C07267=1135.788,-43.089,-47.280,179.177,6.196,149.362
C07268=1135.793,-43.339,-47.268,179.175,6.195,149.362
C07269=1135.798,-43.589,-47.258,179.172,6.194,149.363
C07270=1135.804,-43.838,-47.246,179.170,6.194,149.363
C07271=1135.809,-44.088,-47.235,179.168,6.193,149.364
C07272=1135.814,-44.337,-47.224,179.165,6.193,149.364
C07273=1135.820,-44.587,-47.213,179.163,6.192,149.365
C07274=1135.825,-44.837,-47.202,179.160,6.191,149.366
C07275=1135.829,-45.086,-47.190,179.158,6.191,149.366
C07276=1135.836,-45.336,-47.180,179.156,6.190,149.367
C07277=1135.840,-45.586,-47.168,179.153,6.189,149.367
C07278=1135.845,-45.835,-47.157,179.151,6.189,149.368
C07279=1135.851,-46.085,-47.146,179.149,6.188,149.368
C07280=1135.856,-46.335,-47.135,179.147,6.187,149.369
C07281=1135.861,-46.585,-47.124,179.144,6.187,149.369
C07282=1135.867,-46.834,-47.113,179.143,6.187,149.370
C07283=1135.872,-47.084,-47.102,179.140,6.186,149.370
C07284=1135.877,-47.334,-47.091,179.138,6.186,149.371
C07285=1135.883,-47.584,-47.079,179.136,6.185,149.371
C07286=1135.887,-47.833,-47.068,179.133,6.184,149.372
C07287=1135.893,-48.083,-47.058,179.131,6.183,149.372
C07288=1135.898,-48.333,-47.046,179.129,6.183,149.373
C07289=1135.903,-48.583,-47.036,179.126,6.182,149.374
C07290=1135.909,-48.832,-47.025,179.124,6.181,149.374
C07291=1135.913,-49.081,-47.013,179.121,6.181,149.375
C07292=1135.919,-49.332,-47.002,179.119,6.180,149.375
C07293=1135.924,-49.581,-46.991,179.117,6.179,149.376
C07294=1135.929,-49.831,-46.981,179.115,6.179,149.376
C07295=1135.935,-50.080,-46.970,179.113,6.179,149.377
C07296=1135.940,-50.331,-46.959,179.111,6.178,149.377
C07297=1135.946,-50.602,-46.946,179.108,6.177,149.378
C07298=1135.952,-50.872,-46.935,179.105,6.176,149.379
C07299=1135.957,-51.143,-46.923,179.103,6.176,149.379
C07300=1135.963,-51.413,-46.911,179.100,6.175,149.380
C07301=1135.968,-51.663,-46.900,179.098,6.174,149.380
C07302=1135.973,-51.913,-46.889,179.097,6.174,149.381
C07303=1135.979,-52.162,-46.879,179.094,6.174,149.381
C07304=1135.984,-52.412,-46.867,179.092,6.173,149.382
C07305=1135.990,-52.662,-46.857,179.090,6.172,149.382
C07306=1135.995,-52.912,-46.846,179.087,6.172,149.383
C07307=1136.000,-53.161,-46.835,179.085,6.171,149.384
C07308=1136.005,-53.411,-46.825,179.082,6.171,149.384
C07309=1136.011,-53.660,-46.813,179.080,6.170,149.385
C07310=1136.016,-53.911,-46.803,179.078,6.169,149.385
C07311=1136.021,-54.160,-46.792,179.075,6.169,149.386
C07312=1136.026,-54.410,-46.781,179.074,6.169,149.386
C07313=1136.031,-54.660,-46.770,179.072,6.168,149.387
C07314=1136.037,-54.909,-46.760,179.069,6.167,149.387
C07315=1136.042,-55.159,-46.749,179.067,6.167,149.388
C07316=1136.048,-55.408,-46.737,179.065,6.166,149.388
C07317=1136.053,-55.659,-46.727,179.062,6.165,149.389
C07318=1136.058,-55.908,-46.717,179.060,6.165,149.390
C07319=1136.063,-56.158,-46.705,179.058,6.164,149.390
C07320=1136.069,-56.407,-46.695,179.056,6.164,149.390
C07321=1136.074,-56.658,-46.685,179.054,6.163,149.391
C07322=1136.079,-56.907,-46.674,179.051,6.163,149.392
C07323=1136.084,-57.157,-46.663,179.049,6.162,149.392
C07324=1136.089,-57.406,-46.653,179.047,6.161,149.393
C07325=1136.094,-57.656,-46.642,179.045,6.161,149.393
C07326=1136.100,-57.906,-46.631,179.042,6.160,149.394
C07327=1136.105,-58.156,-46.620,179.040,6.159,149.394
C07328=1136.111,-58.405,-46.609,179.038,6.159,149.395
C07329=1136.116,-58.655,-46.599,179.035,6.159,149.395
C07330=1136.121,-58.905,-46.589,179.033,6.158,149.396
C07331=1136.126,-59.155,-46.578,179.031,6.157,149.396
C07332=1136.132,-59.404,-46.567,179.029,6.157,149.397
C07333=1136.137,-59.654,-46.557,179.026,6.156,149.398
C07334=1136.142,-59.904,-46.546,179.024,6.156,149.398
C07335=1136.148,-60.153,-46.536,179.022,6.156,149.399
C07336=1136.153,-60.403,-46.525,179.020,6.155,149.399
C07337=1136.158,-60.652,-46.515,179.018,6.154,149.400
C07338=1136.163,-60.903,-46.504,179.015,6.154,149.400
C07339=1136.169,-61.152,-46.494,179.013,6.153,149.401
C07340=1136.174,-61.403,-46.483,179.011,6.152,149.401
C07341=1136.179,-61.651,-46.472,179.008,6.152,149.402
C07342=1136.185,-61.901,-46.462,179.007,6.152,149.402
C07343=1136.190,-62.151,-46.451,179.004,6.151,149.403
C07344=1136.195,-62.401,-46.441,179.002,6.150,149.403
C07345=1136.200,-62.651,-46.431,179.000,6.150,149.404
C07346=1136.205,-62.900,-46.420,178.997,6.149,149.405
C07347=1136.211,-63.149,-46.410,178.995,6.148,149.405
C07348=1136.216,-63.400,-46.399,178.994,6.148,149.406
C07349=1136.222,-63.649,-46.389,178.991,6.148,149.406
C07350=1136.227,-63.900,-46.378,178.989,6.147,149.407
C07351=1136.232,-64.149,-46.368,178.987,6.146,149.407
C07352=1136.238,-64.399,-46.358,178.984,6.146,149.408
C07353=1136.243,-64.649,-46.347,178.982,6.145,149.408
C07354=1136.248,-64.898,-46.338,178.980,6.145,149.409
C07355=1136.252,-65.148,-46.326,178.978,6.145,149.409
C07356=1136.258,-65.397,-46.316,178.976,6.144,149.410
C07357=1136.264,-65.647,-46.306,178.974,6.143,149.410
C07358=1136.269,-65.897,-46.295,178.971,6.143,149.411
C07359=1136.274,-66.147,-46.285,178.969,6.142,149.411
C07360=1136.280,-66.396,-46.275,178.967,6.142,149.412
C07361=1136.285,-66.646,-46.264,178.965,6.141,149.412
C07362=1136.290,-66.896,-46.254,178.962,6.141,149.413
C07363=1136.296,-67.145,-46.244,178.960,6.140,149.414
C07364=1136.301,-67.396,-46.233,178.958,6.139,149.414
C07365=1136.306,-67.645,-46.224,178.956,6.139,149.415
C07366=1136.311,-67.894,-46.213,178.954,6.139,149.415
C07367=1136.316,-68.145,-46.203,178.951,6.138,149.416
C07368=1136.322,-68.394,-46.193,178.949,6.137,149.416
C07369=1136.328,-68.644,-46.182,178.947,6.137,149.417
C07370=1136.333,-68.894,-46.172,178.945,6.136,149.417
C07371=1136.338,-69.144,-46.162,178.943,6.136,149.418
C07372=1136.343,-69.393,-46.152,178.941,6.136,149.418
C07373=1136.348,-69.643,-46.142,178.938,6.135,149.419
C07374=1136.354,-69.893,-46.131,178.936,6.134,149.419
C07375=1136.359,-70.142,-46.121,178.933,6.134,149.420
C07376=1136.364,-70.392,-46.111,178.932,6.134,149.421
C07377=1136.370,-70.642,-46.100,178.930,6.133,149.421
C07378=1136.375,-70.891,-46.091,178.928,6.132,149.422
C07379=1136.380,-71.141,-46.081,178.925,6.131,149.422
C07380=1136.386,-71.392,-46.071,178.923,6.132,149.423
C07381=1136.391,-71.641,-46.060,178.921,6.131,149.423
C07382=1136.397,-71.891,-46.050,178.919,6.130,149.424
C07383=1136.401,-72.141,-46.040,178.917,6.129,149.424
C07384=1136.407,-72.390,-46.030,178.914,6.129,149.425
C07385=1136.412,-72.640,-46.020,178.912,6.129,149.425
C07386=1136.418,-72.889,-46.010,178.910,6.128,149.426
C07387=1136.422,-73.139,-46.000,178.908,6.128,149.426
C07388=1136.428,-73.389,-45.990,178.906,6.127,149.427
C07389=1136.434,-73.639,-45.980,178.903,6.126,149.428
C07390=1136.439,-73.888,-45.970,178.902,6.127,149.428
C07391=1136.444,-74.139,-45.959,178.899,6.126,149.428
C07392=1136.449,-74.388,-45.950,178.897,6.125,149.429
C07393=1136.455,-74.637,-45.939,178.895,6.124,149.429
C07394=1136.461,-74.888,-45.930,178.893,6.125,149.430
C07395=1136.465,-75.138,-45.920,178.891,6.124,149.431
C07396=1136.470,-75.387,-45.910,178.889,6.123,149.431
C07397=1136.476,-75.637,-45.899,178.886,6.122,149.432
C07398=1136.482,-75.886,-45.889,178.884,6.122,149.432
C07399=1136.487,-76.136,-45.880,178.882,6.122,149.433
C07400=1136.492,-76.386,-45.870,178.880,6.121,149.433
C07401=1136.498,-76.657,-45.859,178.878,6.120,149.434
C07402=1136.504,-76.929,-45.848,178.875,6.120,149.434
C07403=1136.509,-77.200,-45.837,178.873,6.119,149.435
C07404=1136.516,-77.472,-45.827,178.871,6.119,149.435
C07405=1136.520,-77.722,-45.817,178.869,6.119,149.436
C07406=1136.526,-77.971,-45.807,178.866,6.118,149.437
C07407=1136.531,-78.221,-45.797,178.864,6.118,149.437
C07408=1136.537,-78.471,-45.788,178.862,6.117,149.438
C07409=1136.542,-78.720,-45.777,178.860,6.117,149.438
C07410=1136.548,-78.970,-45.767,178.858,6.116,149.439
C07411=1136.552,-79.220,-45.758,178.856,6.116,149.439
C07412=1136.558,-79.470,-45.748,178.853,6.115,149.440
C07413=1136.563,-79.719,-45.738,178.852,6.115,149.440
C07414=1136.569,-79.969,-45.729,178.850,6.114,149.441
C07415=1136.574,-80.219,-45.718,178.847,6.113,149.441
C07416=1136.580,-80.468,-45.708,178.845,6.113,149.442
C07417=1136.584,-80.719,-45.699,178.843,6.113,149.442
C07418=1136.590,-80.969,-45.689,178.841,6.112,149.443
C07419=1136.595,-81.218,-45.679,178.839,6.112,149.443
C07420=1136.601,-81.468,-45.670,178.836,6.111,149.444
C07421=1136.606,-81.717,-45.659,178.835,6.111,149.444
C07422=1136.612,-81.967,-45.651,178.832,6.110,149.445
C07423=1136.617,-82.218,-45.640,178.830,6.110,149.446
C07424=1136.621,-82.467,-45.630,178.828,6.109,149.446
C07425=1136.627,-82.717,-45.621,178.826,6.109,149.447
C07426=1136.632,-82.966,-45.611,178.824,6.108,149.447
C07427=1136.638,-83.216,-45.602,178.822,6.107,149.447
C07428=1136.644,-83.466,-45.592,178.820,6.108,149.448
C07429=1136.649,-83.716,-45.583,178.818,6.107,149.449
C07430=1136.654,-83.965,-45.572,178.815,6.106,149.449
C07431=1136.659,-84.215,-45.563,178.813,6.106,149.450
C07432=1136.665,-84.465,-45.553,178.812,6.106,149.450
C07433=1136.669,-84.715,-45.543,178.809,6.105,149.451
C07434=1136.675,-84.965,-45.534,178.807,6.105,149.451
C07435=1136.680,-85.214,-45.524,178.805,6.104,149.452
C07436=1136.686,-85.464,-45.515,178.803,6.104,149.452
C07437=1136.691,-85.713,-45.505,178.801,6.103,149.453
C07438=1136.697,-85.964,-45.496,178.799,6.102,149.453
C07439=1136.702,-86.213,-45.486,178.797,6.102,149.454
C07440=1136.708,-86.463,-45.477,178.794,6.102,149.454
C07441=1136.713,-86.712,-45.467,178.792,6.101,149.455
C07442=1136.718,-86.963,-45.457,178.790,6.100,149.455
C07443=1136.723,-87.212,-45.447,178.788,6.100,149.456
C07444=1136.729,-87.462,-45.438,178.786,6.100,149.456
C07445=1136.733,-87.712,-45.428,178.784,6.099,149.457
C07446=1136.739,-87.962,-45.419,178.782,6.099,149.458
C07447=1136.745,-88.212,-45.410,178.780,6.099,149.458
C07448=1136.749,-88.461,-45.400,178.777,6.098,149.459
C07449=1136.755,-88.711,-45.391,178.776,6.098,149.459
C07450=1136.760,-88.960,-45.381,178.774,6.097,149.460
C07451=1136.766,-89.210,-45.372,178.771,6.096,149.460
C07452=1136.771,-89.460,-45.362,178.769,6.096,149.460
C07453=1136.777,-89.710,-45.353,178.767,6.096,149.461
C07454=1136.782,-89.960,-45.344,178.765,6.095,149.462
C07455=1136.788,-90.209,-45.334,178.763,6.095,149.462
C07456=1136.793,-90.459,-45.325,178.761,6.095,149.463
C07457=1136.798,-90.708,-45.315,178.759,6.094,149.463
C07458=1136.803,-90.959,-45.306,178.757,6.093,149.464
C07459=1136.809,-91.208,-45.297,178.755,6.093,149.464
C07460=1136.814,-91.458,-45.286,178.753,6.093,149.465
C07461=1136.819,-91.708,-45.278,178.750,6.092,149.465
C07462=1136.825,-91.958,-45.269,178.749,6.092,149.466
C07463=1136.830,-92.207,-45.258,178.747,6.091,149.466
C07464=1136.835,-92.457,-45.250,178.744,6.091,149.467
C07465=1136.841,-92.707,-45.241,178.743,6.091,149.467
C07466=1136.846,-92.956,-45.230,178.741,6.090,149.468
C07467=1136.851,-93.206,-45.222,178.738,6.089,149.468
C07468=1136.857,-93.456,-45.212,178.736,6.090,149.469
C07469=1136.862,-93.706,-45.203,178.734,6.089,149.469
C07470=1136.867,-93.955,-45.194,178.732,6.088,149.470
C07471=1136.873,-94.206,-45.184,178.730,6.088,149.470
C07472=1136.878,-94.456,-45.175,178.728,6.087,149.471
C07473=1136.883,-94.705,-45.166,178.726,6.087,149.471
C07474=1136.889,-94.955,-45.156,178.724,6.087,149.472
C07475=1136.894,-95.205,-45.147,178.722,6.086,149.473
C07476=1136.899,-95.455,-45.138,178.719,6.085,149.473
C07477=1136.905,-95.704,-45.128,178.718,6.085,149.474
C07478=1136.910,-95.954,-45.119,178.716,6.085,149.474
C07479=1136.915,-96.204,-45.110,178.713,6.084,149.474
C07480=1136.920,-96.454,-45.101,178.712,6.084,149.475
C07481=1136.926,-96.704,-45.092,178.710,6.083,149.475
C07482=1136.931,-96.953,-45.082,178.707,6.083,149.476
C07483=1136.936,-97.203,-45.073,178.706,6.083,149.476
C07484=1136.942,-97.453,-45.064,178.703,6.082,149.477
C07485=1136.948,-97.702,-45.055,178.701,6.081,149.478
C07486=1136.953,-97.952,-45.046,178.699,6.081,149.478
C07487=1136.958,-98.201,-45.037,178.697,6.081,149.479
C07488=1136.964,-98.452,-45.027,178.695,6.080,149.479
C07489=1136.969,-98.701,-45.018,178.693,6.080,149.480
C07490=1136.974,-98.951,-45.010,178.691,6.079,149.480
C07491=1136.980,-99.201,-45.000,178.689,6.079,149.481
C07492=1136.985,-99.451,-44.991,178.687,6.079,149.481
C07493=1136.991,-99.701,-44.982,178.685,6.078,149.482
C07494=1136.996,-99.951,-44.973,178.683,6.077,149.482
C07495=1137.001,-100.200,-44.963,178.681,6.077,149.483
C07496=1137.007,-100.450,-44.955,178.679,6.077,149.483
C07497=1137.012,-100.699,-44.946,178.677,6.077,149.484
C07498=1137.017,-100.949,-44.937,178.675,6.076,149.484
C07499=1137.023,-101.199,-44.928,178.673,6.075,149.485
C07500=1137.029,-101.449,-44.918,178.671,6.075,149.485
C07501=1137.034,-101.699,-44.910,178.669,6.075,149.486
C07502=1137.039,-101.949,-44.901,178.667,6.074,149.486
C07503=1137.044,-102.199,-44.892,178.665,6.074,149.487
C07504=1137.049,-102.449,-44.883,178.663,6.074,149.487
C07505=1137.055,-102.720,-44.873,178.660,6.073,149.488
C07506=1137.062,-102.993,-44.863,178.659,6.073,149.488
C07507=1137.067,-103.265,-44.853,178.657,6.072,149.489
C07508=1137.073,-103.537,-44.843,178.654,6.072,149.489
C07509=1137.078,-103.787,-44.834,178.652,6.071,149.490
C07510=1137.083,-104.037,-44.825,178.650,6.071,149.490
C07511=1137.089,-104.286,-44.817,178.648,6.070,149.491
C07512=1137.094,-104.536,-44.808,178.646,6.070,149.491
C07513=1137.100,-104.786,-44.799,178.644,6.070,149.492
C07514=1137.105,-105.036,-44.789,178.642,6.069,149.492
C07515=1137.111,-105.286,-44.781,178.640,6.069,149.493
C07516=1137.116,-105.536,-44.772,178.638,6.068,149.493
C07517=1137.121,-105.786,-44.763,178.636,6.067,149.494
C07518=1137.127,-106.035,-44.754,178.634,6.067,149.494
C07519=1137.132,-106.285,-44.745,178.632,6.067,149.495
C07520=1137.137,-106.534,-44.736,178.631,6.067,149.495
C07521=1137.142,-106.784,-44.728,178.628,6.066,149.496
C07522=1137.147,-107.034,-44.719,178.626,6.066,149.497
C07523=1137.153,-107.283,-44.710,178.624,6.066,149.497
C07524=1137.159,-107.533,-44.701,178.622,6.065,149.497
C07525=1137.165,-107.784,-44.692,178.620,6.065,149.498
C07526=1137.170,-108.034,-44.684,178.618,6.064,149.498
C07527=1137.175,-108.284,-44.675,178.616,6.063,149.499
C07528=1137.181,-108.533,-44.666,178.614,6.063,149.499
C07529=1137.186,-108.783,-44.657,178.612,6.063,149.500
C07530=1137.191,-109.032,-44.648,178.610,6.063,149.500
C07531=1137.196,-109.282,-44.639,178.608,6.062,149.501
C07532=1137.201,-109.532,-44.631,178.606,6.061,149.501
C07533=1137.207,-109.781,-44.622,178.604,6.061,149.502
C07534=1137.213,-110.032,-44.614,178.602,6.061,149.502
C07535=1137.218,-110.282,-44.605,178.601,6.061,149.503
C07536=1137.223,-110.531,-44.596,178.598,6.060,149.503
C07537=1137.229,-110.781,-44.588,178.597,6.060,149.504
C07538=1137.234,-111.030,-44.579,178.595,6.059,149.504
C07539=1137.239,-111.280,-44.570,178.592,6.058,149.505
C07540=1137.244,-111.530,-44.561,178.590,6.059,149.506
C07541=1137.250,-111.780,-44.553,178.588,6.058,149.506
C07542=1137.255,-112.030,-44.544,178.587,6.058,149.506
C07543=1137.261,-112.280,-44.535,178.584,6.057,149.507
C07544=1137.266,-112.530,-44.526,178.582,6.057,149.507
C07545=1137.271,-112.779,-44.518,178.581,6.057,149.508
C07546=1137.277,-113.029,-44.510,178.578,6.056,149.508
C07547=1137.282,-113.279,-44.501,178.577,6.056,149.509
C07548=1137.287,-113.529,-44.492,178.575,6.055,149.509
C07549=1137.293,-113.778,-44.483,178.573,6.055,149.510
C07550=1137.299,-114.028,-44.475,178.571,6.055,149.510
C07551=1137.304,-114.278,-44.466,178.569,6.054,149.511
C07552=1137.309,-114.527,-44.458,178.567,6.054,149.511
C07553=1137.315,-114.777,-44.449,178.565,6.053,149.512
C07554=1137.320,-115.028,-44.441,178.563,6.053,149.512
C07555=1137.325,-115.278,-44.432,178.561,6.052,149.513
C07556=1137.331,-115.527,-44.423,178.559,6.052,149.513
C07557=1137.336,-115.777,-44.414,178.557,6.052,149.514
C07558=1137.342,-116.027,-44.406,178.555,6.051,149.514
C07559=1137.347,-116.276,-44.398,178.553,6.051,149.515
C07560=1137.353,-116.526,-44.389,178.551,6.050,149.515
C07561=1137.358,-116.777,-44.380,178.550,6.050,149.516
C07562=1137.364,-117.026,-44.372,178.547,6.050,149.516
C07563=1137.369,-117.276,-44.363,178.546,6.050,149.517
C07564=1137.374,-117.526,-44.355,178.544,6.049,149.517
C07565=1137.380,-117.775,-44.347,178.542,6.049,149.518
C07566=1137.385,-118.025,-44.338,178.540,6.048,149.518
C07567=1137.390,-118.275,-44.330,178.538,6.047,149.519
C07568=1137.396,-118.524,-44.321,178.536,6.047,149.519
C07569=1137.401,-118.774,-44.312,178.534,6.047,149.520
C07570=1137.407,-119.025,-44.304,178.532,6.047,149.520
C07571=1137.412,-119.274,-44.296,178.530,6.046,149.521
C07572=1137.417,-119.524,-44.287,178.529,6.046,149.521
C07573=1137.422,-119.774,-44.279,178.526,6.045,149.522
C07574=1137.428,-120.023,-44.271,178.525,6.045,149.522
C07575=1137.433,-120.273,-44.262,178.523,6.045,149.523
C07576=1137.439,-120.523,-44.254,178.521,6.045,149.523
C07577=1137.444,-120.772,-44.245,178.519,6.044,149.524
C07578=1137.450,-121.023,-44.237,178.517,6.043,149.524
C07579=1137.456,-121.272,-44.228,178.515,6.043,149.525
C07580=1137.460,-121.522,-44.221,178.513,6.042,149.525
C07581=1137.466,-121.772,-44.212,178.511,6.042,149.525
C07582=1137.471,-122.021,-44.203,178.509,6.042,149.526
C07583=1137.477,-122.272,-44.195,178.507,6.042,149.526
C07584=1137.482,-122.522,-44.186,178.505,6.041,149.527
C07585=1137.487,-122.771,-44.179,178.504,6.041,149.527
C07586=1137.492,-123.021,-44.170,178.501,6.040,149.528
C07587=1137.499,-123.271,-44.162,178.500,6.040,149.528
C07588=1137.504,-123.520,-44.153,178.498,6.040,149.529
C07589=1137.509,-123.771,-44.145,178.496,6.040,149.529
C07590=1137.514,-124.020,-44.137,178.494,6.039,149.530
C07591=1137.520,-124.270,-44.129,178.492,6.039,149.530
C07592=1137.525,-124.519,-44.121,178.490,6.038,149.531
C07593=1137.531,-124.770,-44.112,178.488,6.038,149.531
C07594=1137.536,-125.020,-44.103,178.486,6.038,149.532
C07595=1137.541,-125.269,-44.096,178.484,6.037,149.532
C07596=1137.547,-125.519,-44.087,178.482,6.037,149.533
C07597=1137.553,-125.769,-44.080,178.481,6.036,149.533
C07598=1137.558,-126.019,-44.071,178.479,6.036,149.534
C07599=1137.563,-126.269,-44.063,178.477,6.035,149.534
C07600=1137.568,-126.518,-44.055,178.475,6.035,149.535
C07601=1137.574,-126.768,-44.046,178.473,6.034,149.535
C07602=1137.580,-127.018,-44.038,178.471,6.034,149.535
C07603=1137.584,-127.268,-44.030,178.469,6.034,149.536
C07604=1137.590,-127.518,-44.022,178.468,6.034,149.536
C07605=1137.596,-127.767,-44.014,178.465,6.033,149.537
C07606=1137.601,-128.017,-44.006,178.464,6.033,149.537
C07607=1137.606,-128.267,-43.997,178.462,6.032,149.538
C07608=1137.612,-128.516,-43.990,178.460,6.032,149.538
C07609=1137.190,-128.528,-44.033,178.456,6.036,149.540
C07610=1137.186,-128.278,-44.041,178.458,6.036,149.540
C07611=1137.180,-128.029,-44.049,178.460,6.036,149.539
C07612=1137.174,-127.778,-44.058,178.462,6.037,149.539
C07613=1137.169,-127.528,-44.066,178.464,6.037,149.538
C07614=1137.164,-127.279,-44.074,178.466,6.038,149.538
C07615=1137.158,-127.029,-44.082,178.468,6.038,149.537
C07616=1137.153,-126.780,-44.090,178.470,6.038,149.537
C07617=1137.147,-126.529,-44.099,178.471,6.038,149.536
C07618=1137.142,-126.280,-44.107,178.474,6.039,149.536
C07619=1137.137,-126.030,-44.115,178.475,6.039,149.535
C07620=1137.132,-125.780,-44.124,178.477,6.040,149.535
C07621=1137.125,-125.530,-44.131,178.479,6.040,149.534
C07622=1137.121,-125.281,-44.140,178.481,6.041,149.534
C07623=1137.115,-125.031,-44.148,178.483,6.040,149.533
C07624=1137.110,-124.780,-44.156,178.485,6.041,149.533
C07625=1137.104,-124.531,-44.164,178.487,6.042,149.532
C07626=1137.099,-124.281,-44.172,178.489,6.042,149.532
C07627=1137.094,-124.031,-44.181,178.491,6.043,149.531
C07628=1137.088,-123.782,-44.189,178.493,6.043,149.531
C07629=1137.083,-123.532,-44.198,178.494,6.044,149.531
C07630=1137.077,-123.282,-44.206,178.496,6.044,149.530
C07631=1137.072,-123.032,-44.214,178.498,6.044,149.530
C07632=1137.067,-122.782,-44.223,178.500,6.044,149.529
C07633=1137.061,-122.533,-44.230,178.502,6.045,149.529
C07634=1137.056,-122.283,-44.239,178.504,6.045,149.528
C07635=1137.050,-122.033,-44.247,178.506,6.046,149.528
C07636=1137.045,-121.784,-44.255,178.507,6.046,149.527
C07637=1137.040,-121.533,-44.264,178.510,6.047,149.527
C07638=1137.034,-121.284,-44.272,178.511,6.046,149.526
C07639=1137.029,-121.034,-44.281,178.513,6.047,149.526
C07640=1137.023,-120.784,-44.289,178.516,6.048,149.525
C07641=1137.018,-120.534,-44.298,178.517,6.048,149.525
C07642=1137.013,-120.284,-44.305,178.519,6.049,149.524
C07643=1137.008,-120.034,-44.314,178.521,6.049,149.524
C07644=1137.002,-119.785,-44.323,178.523,6.049,149.523
C07645=1136.996,-119.535,-44.331,178.525,6.049,149.523
C07646=1136.991,-119.286,-44.339,178.527,6.050,149.522
C07647=1136.985,-119.035,-44.348,178.528,6.050,149.522
C07648=1136.980,-118.785,-44.357,178.531,6.051,149.521
C07649=1136.975,-118.536,-44.364,178.532,6.051,149.521
C07650=1136.969,-118.286,-44.373,178.534,6.051,149.520
C07651=1136.964,-118.036,-44.382,178.537,6.052,149.520
C07652=1136.959,-117.787,-44.390,178.538,6.052,149.519
C07653=1136.953,-117.537,-44.398,178.540,6.053,149.519
C07654=1136.948,-117.287,-44.407,178.542,6.053,149.519
C07655=1136.942,-117.038,-44.416,178.544,6.054,149.518
C07656=1136.937,-116.787,-44.424,178.546,6.054,149.518
C07657=1136.932,-116.537,-44.433,178.548,6.054,149.517
C07658=1136.926,-116.287,-44.442,178.550,6.054,149.517
C07659=1136.920,-116.038,-44.449,178.552,6.055,149.516
C07660=1136.916,-115.788,-44.458,178.554,6.056,149.516
C07661=1136.911,-115.538,-44.467,178.556,6.056,149.515
C07662=1136.905,-115.289,-44.475,178.558,6.056,149.515
C07663=1136.899,-115.039,-44.483,178.559,6.056,149.514
C07664=1136.894,-114.789,-44.492,178.562,6.057,149.514
C07665=1136.889,-114.540,-44.501,178.563,6.057,149.513
C07666=1136.883,-114.289,-44.509,178.565,6.058,149.513
C07667=1136.878,-114.039,-44.518,178.568,6.059,149.512
C07668=1136.873,-113.789,-44.527,178.569,6.059,149.512
C07669=1136.867,-113.540,-44.535,178.571,6.059,149.511
C07670=1136.861,-113.290,-44.544,178.573,6.059,149.511
C07671=1136.856,-113.040,-44.552,178.575,6.060,149.510
C07672=1136.851,-112.791,-44.561,178.577,6.060,149.510
C07673=1136.845,-112.541,-44.570,178.579,6.061,149.509
C07674=1136.840,-112.291,-44.579,178.581,6.061,149.509
C07675=1136.835,-112.041,-44.587,178.583,6.061,149.508
C07676=1136.829,-111.791,-44.595,178.585,6.062,149.508
C07677=1136.824,-111.542,-44.604,178.587,6.062,149.507
C07678=1136.819,-111.292,-44.613,178.589,6.062,149.507
C07679=1136.813,-111.042,-44.622,178.591,6.062,149.506
C07680=1136.808,-110.793,-44.631,178.593,6.063,149.506
C07681=1136.802,-110.542,-44.639,178.595,6.064,149.505
C07682=1136.797,-110.292,-44.648,178.597,6.064,149.505
C07683=1136.792,-110.043,-44.657,178.599,6.065,149.504
C07684=1136.786,-109.793,-44.665,178.601,6.065,149.504
C07685=1136.781,-109.544,-44.674,178.603,6.065,149.503
C07686=1136.776,-109.294,-44.683,178.605,6.066,149.503
C07687=1136.771,-109.044,-44.692,178.607,6.066,149.502
C07688=1136.765,-108.793,-44.700,178.609,6.067,149.502
C07689=1136.759,-108.544,-44.709,178.610,6.067,149.501
C07690=1136.753,-108.294,-44.718,178.613,6.067,149.501
C07691=1136.748,-108.044,-44.727,178.615,6.068,149.500
C07692=1136.743,-107.794,-44.736,178.616,6.068,149.500
C07693=1136.737,-107.545,-44.744,178.619,6.069,149.499
C07694=1136.732,-107.295,-44.753,178.620,6.069,149.499
C07695=1136.727,-107.046,-44.762,178.622,6.070,149.498
C07696=1136.722,-106.796,-44.771,178.625,6.070,149.498
C07697=1136.717,-106.546,-44.780,178.626,6.070,149.497
C07698=1136.712,-106.296,-44.789,178.629,6.071,149.497
C07699=1136.706,-106.047,-44.797,178.630,6.071,149.496
C07700=1136.700,-105.797,-44.807,178.633,6.071,149.496
C07701=1136.695,-105.547,-44.816,178.635,6.072,149.495
C07702=1136.690,-105.297,-44.825,178.636,6.072,149.495
C07703=1136.684,-105.047,-44.834,178.639,6.073,149.494
C07704=1136.679,-104.797,-44.842,178.641,6.074,149.494
C07705=1136.673,-104.548,-44.850,178.642,6.074,149.493
C07706=1136.668,-104.298,-44.859,178.645,6.074,149.493
C07707=1136.663,-104.048,-44.869,178.646,6.074,149.492
C07708=1136.657,-103.798,-44.878,178.648,6.075,149.492
C07709=1136.652,-103.548,-44.887,178.651,6.076,149.491
C07710=1136.646,-103.276,-44.897,178.653,6.075,149.491
C07711=1136.640,-103.004,-44.906,178.655,6.076,149.490
C07712=1136.634,-102.732,-44.916,178.657,6.077,149.490
C07713=1136.629,-102.460,-44.926,178.659,6.078,149.489
C07714=1136.623,-102.210,-44.935,178.661,6.078,149.489
C07715=1136.618,-101.960,-44.943,178.664,6.078,149.488
C07716=1136.612,-101.710,-44.953,178.666,6.079,149.487
C07717=1136.607,-101.460,-44.962,178.667,6.079,149.487
C07718=1136.602,-101.210,-44.971,178.670,6.079,149.486
C07719=1136.596,-100.961,-44.979,178.671,6.079,149.486
C07720=1136.591,-100.712,-44.989,178.673,6.080,149.485
C07721=1136.585,-100.461,-44.998,178.676,6.081,149.485
C07722=1136.580,-100.212,-45.007,178.677,6.081,149.485
C07723=1136.575,-99.962,-45.016,178.679,6.082,149.484
C07724=1136.570,-99.712,-45.025,178.682,6.082,149.484
C07725=1136.564,-99.462,-45.035,178.683,6.082,149.483
C07726=1136.559,-99.212,-45.043,178.686,6.083,149.482
C07727=1136.554,-98.962,-45.052,178.688,6.083,149.482
C07728=1136.548,-98.714,-45.062,178.690,6.083,149.481
C07729=1136.542,-98.463,-45.071,178.692,6.084,149.481
C07730=1136.537,-98.213,-45.080,178.694,6.085,149.480
C07731=1136.532,-97.964,-45.089,178.696,6.085,149.480
C07732=1136.527,-97.714,-45.098,178.698,6.085,149.479
C07733=1136.521,-97.464,-45.107,178.700,6.086,149.479
C07734=1136.516,-97.214,-45.117,178.702,6.086,149.478
C07735=1136.511,-96.965,-45.126,178.704,6.087,149.478
C07736=1136.505,-96.714,-45.135,178.706,6.087,149.477
C07737=1136.500,-96.465,-45.144,178.708,6.087,149.477
C07738=1136.495,-96.215,-45.153,178.710,6.088,149.476
C07739=1136.490,-95.965,-45.163,178.712,6.088,149.476
C07740=1136.484,-95.715,-45.172,178.714,6.089,149.475
C07741=1136.479,-95.465,-45.181,178.716,6.089,149.475
C07742=1136.474,-95.216,-45.190,178.718,6.089,149.474
C07743=1136.467,-94.967,-45.200,178.720,6.090,149.474
C07744=1136.462,-94.717,-45.209,178.722,6.091,149.473
C07745=1136.457,-94.467,-45.218,178.724,6.091,149.473
C07746=1136.451,-94.217,-45.227,178.726,6.091,149.472
C07747=1136.446,-93.968,-45.237,178.729,6.092,149.472
C07748=1136.441,-93.718,-45.246,178.730,6.092,149.471
C07749=1136.435,-93.468,-45.255,178.732,6.093,149.471
C07750=1136.430,-93.218,-45.264,178.735,6.094,149.470
C07751=1136.425,-92.969,-45.274,178.736,6.093,149.470
C07752=1136.419,-92.718,-45.283,178.738,6.094,149.469
C07753=1136.414,-92.469,-45.292,178.741,6.095,149.469
C07754=1136.409,-92.219,-45.302,178.743,6.095,149.468
C07755=1136.403,-91.969,-45.311,178.745,6.095,149.468
C07756=1136.398,-91.719,-45.320,178.747,6.096,149.467
C07757=1136.393,-91.470,-45.330,178.749,6.097,149.467
C07758=1136.387,-91.220,-45.339,178.751,6.097,149.466
C07759=1136.382,-90.970,-45.349,178.753,6.098,149.466
C07760=1136.377,-90.720,-45.358,178.755,6.098,149.465
C07761=1136.371,-90.471,-45.367,178.757,6.098,149.464
C07762=1136.366,-90.220,-45.377,178.760,6.099,149.464
C07763=1136.361,-89.971,-45.386,178.762,6.099,149.463
C07764=1136.355,-89.721,-45.396,178.763,6.099,149.463
C07765=1136.350,-89.472,-45.405,178.766,6.100,149.463
C07766=1136.345,-89.221,-45.415,178.768,6.101,149.462
C07767=1136.339,-88.971,-45.424,178.769,6.101,149.462
C07768=1136.335,-88.722,-45.434,178.772,6.101,149.461
C07769=1136.329,-88.472,-45.443,178.774,6.102,149.460
C07770=1136.324,-88.223,-45.453,178.776,6.103,149.460
C07771=1136.318,-87.972,-45.462,178.778,6.103,149.459
C07772=1136.313,-87.723,-45.472,178.780,6.103,149.459
C07773=1136.307,-87.473,-45.481,178.782,6.104,149.458
C07774=1136.302,-87.224,-45.491,178.784,6.104,149.458
C07775=1136.297,-86.974,-45.500,178.787,6.104,149.457
C07776=1136.291,-86.724,-45.509,178.789,6.105,149.457
C07777=1136.286,-86.474,-45.519,178.791,6.106,149.456
C07778=1136.280,-86.224,-45.529,178.793,6.106,149.456
C07779=1136.276,-85.975,-45.538,178.795,6.107,149.455
C07780=1136.270,-85.725,-45.548,178.797,6.107,149.455
C07781=1136.265,-85.475,-45.558,178.799,6.107,149.454
C07782=1136.260,-85.225,-45.567,178.801,6.108,149.454
C07783=1136.255,-84.976,-45.577,178.804,6.109,149.453
C07784=1136.249,-84.725,-45.586,178.806,6.109,149.453
C07785=1136.244,-84.476,-45.596,178.807,6.109,149.452
C07786=1136.238,-84.227,-45.606,178.809,6.110,149.452
C07787=1136.232,-83.976,-45.616,178.812,6.110,149.451
C07788=1136.228,-83.727,-45.625,178.814,6.110,149.450
C07789=1136.222,-83.477,-45.635,178.816,6.111,149.450
C07790=1136.217,-83.228,-45.644,178.818,6.112,149.450
C07791=1136.212,-82.977,-45.654,178.820,6.113,149.449
C07792=1136.207,-82.728,-45.664,178.822,6.113,149.449
C07793=1136.201,-82.478,-45.674,178.825,6.113,149.448
C07794=1136.196,-82.228,-45.683,178.827,6.114,149.447
C07795=1136.190,-81.979,-45.693,178.829,6.114,149.447
C07796=1136.184,-81.729,-45.703,178.831,6.114,149.446
C07797=1136.180,-81.479,-45.712,178.833,6.115,149.446
C07798=1136.175,-81.229,-45.723,178.835,6.116,149.445
C07799=1136.169,-80.979,-45.732,178.837,6.116,149.445
C07800=1136.164,-80.730,-45.742,178.839,6.116,149.444
C07801=1136.158,-80.480,-45.751,178.841,6.117,149.444
C07802=1136.153,-80.230,-45.761,178.844,6.118,149.443
C07803=1136.147,-79.981,-45.771,178.845,6.118,149.443
C07804=1136.142,-79.731,-45.780,178.847,6.119,149.442
C07805=1136.137,-79.481,-45.791,178.850,6.119,149.442
C07806=1136.132,-79.231,-45.801,178.852,6.120,149.441
C07807=1136.126,-78.981,-45.810,178.854,6.120,149.441
C07808=1136.121,-78.732,-45.820,178.856,6.120,149.440
C07809=1136.115,-78.482,-45.830,178.858,6.121,149.440
C07810=1136.111,-78.232,-45.840,178.861,6.122,149.439
C07811=1136.105,-77.982,-45.850,178.863,6.122,149.438
C07812=1136.100,-77.733,-45.860,178.865,6.122,149.438
C07813=1136.095,-77.483,-45.869,178.867,6.123,149.437
C07814=1136.088,-77.211,-45.880,178.870,6.123,149.437
C07815=1136.083,-76.941,-45.891,178.872,6.124,149.436
C07816=1136.076,-76.668,-45.902,178.874,6.125,149.436
C07817=1136.071,-76.397,-45.913,178.877,6.125,149.435
C07818=1136.066,-76.148,-45.923,178.878,6.125,149.435
C07819=1136.060,-75.898,-45.932,178.880,6.126,149.434
C07820=1136.055,-75.647,-45.942,178.883,6.127,149.434
C07821=1136.050,-75.398,-45.952,178.885,6.128,149.433
C07822=1136.044,-75.148,-45.963,178.887,6.127,149.432
C07823=1136.039,-74.899,-45.972,178.889,6.128,149.432
C07824=1136.033,-74.649,-45.982,178.891,6.129,149.431
C07825=1136.028,-74.399,-45.992,178.893,6.129,149.431
C07826=1136.023,-74.149,-46.003,178.896,6.130,149.431
C07827=1136.018,-73.900,-46.012,178.898,6.130,149.430
C07828=1136.012,-73.650,-46.022,178.900,6.130,149.429
C07829=1136.007,-73.400,-46.033,178.902,6.131,149.429
C07830=1136.002,-73.150,-46.042,178.904,6.132,149.428
C07831=1135.997,-72.901,-46.052,178.906,6.132,149.428
C07832=1135.991,-72.651,-46.062,178.909,6.132,149.427
C07833=1135.986,-72.401,-46.073,178.911,6.133,149.427
C07834=1135.980,-72.151,-46.083,178.913,6.134,149.426
C07835=1135.976,-71.902,-46.093,178.915,6.135,149.426
C07836=1135.970,-71.653,-46.103,178.917,6.134,149.425
C07837=1135.965,-71.402,-46.113,178.919,6.135,149.425
C07838=1135.959,-71.152,-46.123,178.922,6.136,149.424
C07839=1135.954,-70.903,-46.133,178.924,6.137,149.424
C07840=1135.949,-70.653,-46.143,178.926,6.137,149.423
C07841=1135.944,-70.403,-46.153,178.928,6.137,149.422
C07842=1135.938,-70.154,-46.164,178.930,6.138,149.422
C07843=1135.932,-69.904,-46.174,178.932,6.138,149.421
C07844=1135.927,-69.654,-46.184,178.935,6.139,149.421
C07845=1135.922,-69.404,-46.195,178.937,6.140,149.420
C07846=1135.917,-69.155,-46.204,178.939,6.139,149.420
C07847=1135.912,-68.905,-46.215,178.941,6.140,149.419
C07848=1135.906,-68.655,-46.225,178.943,6.141,149.419
C07849=1135.901,-68.406,-46.235,178.946,6.142,149.418
C07850=1135.896,-68.156,-46.246,178.948,6.142,149.418
C07851=1135.890,-67.906,-46.256,178.950,6.142,149.417
C07852=1135.885,-67.656,-46.266,178.952,6.143,149.417
C07853=1135.880,-67.406,-46.276,178.954,6.144,149.416
C07854=1135.875,-67.157,-46.286,178.956,6.144,149.416
C07855=1135.869,-66.907,-46.297,178.959,6.145,149.415
C07856=1135.864,-66.657,-46.307,178.961,6.146,149.414
C07857=1135.859,-66.408,-46.317,178.963,6.146,149.414
C07858=1135.853,-66.158,-46.328,178.965,6.146,149.414
C07859=1135.848,-65.908,-46.338,178.968,6.147,149.413
C07860=1135.842,-65.658,-46.348,178.970,6.147,149.412
C07861=1135.837,-65.409,-46.359,178.972,6.148,149.412
C07862=1135.832,-65.158,-46.369,178.974,6.148,149.411
C07863=1135.826,-64.909,-46.379,178.976,6.149,149.411
C07864=1135.822,-64.659,-46.389,178.978,6.149,149.410
C07865=1135.817,-64.410,-46.400,178.981,6.150,149.410
C07866=1135.811,-64.161,-46.410,178.983,6.151,149.409
C07867=1135.806,-63.910,-46.421,178.985,6.152,149.409
C07868=1135.800,-63.661,-46.431,178.987,6.151,149.408
C07869=1135.795,-63.411,-46.441,178.989,6.152,149.408
C07870=1135.790,-63.161,-46.452,178.992,6.153,149.407
C07871=1135.784,-62.911,-46.462,178.994,6.154,149.407
C07872=1135.779,-62.661,-46.473,178.996,6.154,149.406
C07873=1135.774,-62.412,-46.484,178.999,6.155,149.405
C07874=1135.769,-62.162,-46.494,179.000,6.155,149.405
C07875=1135.763,-61.912,-46.504,179.002,6.155,149.404
C07876=1135.758,-61.663,-46.515,179.005,6.156,149.404
C07877=1135.753,-61.413,-46.525,179.007,6.157,149.403
C07878=1135.747,-61.164,-46.536,179.009,6.157,149.403
C07879=1135.742,-60.914,-46.547,179.012,6.158,149.402
C07880=1135.737,-60.664,-46.557,179.014,6.158,149.402
C07881=1135.732,-60.414,-46.568,179.016,6.158,149.401
C07882=1135.726,-60.164,-46.578,179.018,6.159,149.401
C07883=1135.721,-59.915,-46.589,179.020,6.160,149.400
C07884=1135.716,-59.665,-46.599,179.023,6.160,149.399
C07885=1135.710,-59.415,-46.609,179.025,6.161,149.399
C07886=1135.705,-59.165,-46.620,179.027,6.162,149.398
C07887=1135.700,-58.916,-46.631,179.030,6.163,149.398
C07888=1135.695,-58.666,-46.642,179.032,6.162,149.397
C07889=1135.689,-58.417,-46.652,179.034,6.163,149.397
C07890=1135.684,-58.166,-46.662,179.036,6.164,149.396
C07891=1135.679,-57.917,-46.673,179.038,6.165,149.396
C07892=1135.674,-57.667,-46.684,179.041,6.165,149.395
C07893=1135.668,-57.417,-46.695,179.043,6.166,149.395
C07894=1135.663,-57.168,-46.706,179.045,6.166,149.394
C07895=1135.658,-56.918,-46.716,179.047,6.167,149.394
C07896=1135.653,-56.668,-46.727,179.049,6.167,149.393
C07897=1135.647,-56.419,-46.738,179.052,6.168,149.393
C07898=1135.642,-56.169,-46.748,179.054,6.168,149.392
C07899=1135.637,-55.919,-46.758,179.056,6.169,149.392
C07900=1135.632,-55.669,-46.770,179.059,6.170,149.391
C07901=1135.626,-55.420,-46.780,179.061,6.170,149.390
C07902=1135.621,-55.170,-46.790,179.063,6.171,149.390
C07903=1135.615,-54.920,-46.802,179.065,6.172,149.389
C07904=1135.610,-54.670,-46.813,179.067,6.171,149.389
C07905=1135.605,-54.421,-46.823,179.070,6.172,149.388
C07906=1135.600,-54.171,-46.834,179.072,6.173,149.388
C07907=1135.594,-53.922,-46.844,179.074,6.173,149.387
C07908=1135.590,-53.672,-46.856,179.077,6.174,149.387
C07909=1135.583,-53.422,-46.866,179.079,6.175,149.386
C07910=1135.579,-53.172,-46.878,179.081,6.176,149.386
C07911=1135.573,-52.923,-46.888,179.084,6.176,149.385
C07912=1135.568,-52.673,-46.899,179.086,6.177,149.384
C07913=1135.563,-52.423,-46.910,179.088,6.178,149.384
C07914=1135.558,-52.174,-46.921,179.090,6.178,149.383
C07915=1135.552,-51.924,-46.932,179.092,6.178,149.383
C07916=1135.547,-51.674,-46.942,179.094,6.179,149.382
C07917=1135.542,-51.424,-46.953,179.097,6.180,149.382
C07918=1135.536,-51.154,-46.965,179.099,6.180,149.381
C07919=1135.530,-50.883,-46.977,179.101,6.181,149.381
C07920=1135.525,-50.612,-46.988,179.104,6.181,149.380
C07921=1135.519,-50.342,-47.000,179.106,6.182,149.379
C07922=1135.514,-50.092,-47.012,179.109,6.183,149.379
C07923=1135.508,-49.841,-47.023,179.111,6.183,149.378
C07924=1135.503,-49.592,-47.034,179.113,6.184,149.378
C07925=1135.498,-49.342,-47.044,179.116,6.185,149.377
C07926=1135.493,-49.093,-47.055,179.118,6.185,149.377
C07927=1135.487,-48.843,-47.066,179.120,6.186,149.376
C07928=1135.482,-48.593,-47.078,179.123,6.186,149.376
C07929=1135.477,-48.344,-47.089,179.125,6.187,149.375
C07930=1135.471,-48.094,-47.100,179.128,6.188,149.374
C07931=1135.466,-47.845,-47.111,179.130,6.188,149.374
C07932=1135.461,-47.594,-47.121,179.132,6.189,149.374
C07933=1135.456,-47.345,-47.133,179.133,6.189,149.373
C07934=1135.450,-47.096,-47.144,179.136,6.190,149.372
C07935=1135.445,-46.845,-47.155,179.138,6.190,149.372
C07936=1135.441,-46.596,-47.166,179.141,6.191,149.371
C07937=1135.435,-46.346,-47.177,179.143,6.191,149.371
C07938=1135.430,-46.096,-47.188,179.145,6.192,149.370
C07939=1135.424,-45.847,-47.199,179.148,6.193,149.370
C07940=1135.419,-45.597,-47.210,179.150,6.194,149.369
C07941=1135.414,-45.347,-47.221,179.152,6.194,149.369
C07942=1135.409,-45.098,-47.232,179.155,6.195,149.368
C07943=1135.403,-44.848,-47.244,179.157,6.196,149.368
C07944=1135.398,-44.598,-47.255,179.159,6.196,149.367
C07945=1135.392,-44.349,-47.266,179.162,6.197,149.366
C07946=1135.388,-44.099,-47.278,179.164,6.198,149.366
C07947=1135.383,-43.849,-47.288,179.166,6.198,149.365
C07948=1135.377,-43.600,-47.300,179.169,6.199,149.365
C07949=1135.372,-43.350,-47.311,179.171,6.200,149.364
C07950=1135.367,-43.100,-47.322,179.173,6.200,149.364
C07951=1135.361,-42.850,-47.333,179.175,6.200,149.363
C07952=1135.356,-42.601,-47.344,179.177,6.201,149.363
C07953=1135.351,-42.351,-47.356,179.180,6.202,149.362
C07954=1135.346,-42.101,-47.368,179.182,6.202,149.362
C07955=1135.340,-41.852,-47.378,179.184,6.203,149.361
C07956=1135.335,-41.602,-47.390,179.187,6.203,149.360
C07957=1135.330,-41.352,-47.401,179.189,6.204,149.360
C07958=1135.325,-41.102,-47.413,179.191,6.205,149.359
C07959=1135.320,-40.853,-47.424,179.194,6.205,149.359
C07960=1135.314,-40.603,-47.435,179.196,6.206,149.358
C07961=1135.309,-40.353,-47.446,179.198,6.207,149.358
C07962=1135.303,-40.104,-47.458,179.201,6.207,149.357
C07963=1135.298,-39.854,-47.469,179.203,6.208,149.357
C07964=1135.293,-39.604,-47.481,179.205,6.209,149.356
C07965=1135.288,-39.355,-47.492,179.208,6.209,149.356
C07966=1135.282,-39.105,-47.503,179.210,6.210,149.355
C07967=1135.277,-38.855,-47.514,179.212,6.211,149.355
C07968=1135.272,-38.605,-47.526,179.215,6.211,149.354
C07969=1135.267,-38.356,-47.537,179.217,6.212,149.353
C07970=1135.261,-38.107,-47.549,179.219,6.213,149.353
C07971=1135.256,-37.857,-47.560,179.222,6.213,149.352
C07972=1135.251,-37.607,-47.572,179.224,6.214,149.352
C07973=1135.246,-37.357,-47.583,179.226,6.215,149.351
C07974=1135.240,-37.108,-47.595,179.228,6.216,149.351
C07975=1135.236,-36.858,-47.606,179.231,6.216,149.350
C07976=1135.230,-36.609,-47.618,179.233,6.217,149.350
C07977=1135.225,-36.358,-47.629,179.235,6.218,149.349
C07978=1135.220,-36.108,-47.641,179.238,6.218,149.348
C07979=1135.214,-35.859,-47.651,179.240,6.219,149.348
C07980=1135.209,-35.609,-47.663,179.242,6.219,149.347
C07981=1135.204,-35.360,-47.675,179.245,6.220,149.347
C07982=1135.199,-35.110,-47.687,179.247,6.221,149.346
C07983=1135.193,-34.860,-47.698,179.249,6.221,149.346
C07984=1135.188,-34.611,-47.709,179.252,6.222,149.345
C07985=1135.183,-34.361,-47.721,179.254,6.223,149.345
C07986=1135.177,-34.111,-47.733,179.256,6.223,149.344
C07987=1135.173,-33.862,-47.744,179.259,6.224,149.344
C07988=1135.167,-33.612,-47.756,179.261,6.225,149.343
C07989=1135.162,-33.362,-47.768,179.264,6.225,149.343
C07990=1135.157,-33.113,-47.780,179.266,6.226,149.342
C07991=1135.151,-32.863,-47.792,179.268,6.227,149.341
C07992=1135.147,-32.614,-47.803,179.271,6.227,149.341
C07993=1135.141,-32.364,-47.815,179.273,6.228,149.340
C07994=1135.136,-32.114,-47.827,179.275,6.228,149.340
C07995=1135.131,-31.864,-47.838,179.278,6.229,149.339
C07996=1135.126,-31.614,-47.850,179.280,6.230,149.339
C07997=1135.120,-31.365,-47.861,179.282,6.230,149.338
C07998=1135.115,-31.116,-47.873,179.285,6.231,149.338
C07999=1135.110,-30.866,-47.885,179.287,6.232,149.337
C08000=1135.104,-30.616,-47.897,179.289,6.232,149.336
C08001=1135.100,-30.367,-47.909,179.292,6.233,149.336
C08002=1135.094,-30.117,-47.920,179.294,6.234,149.335
C08003=1135.089,-29.867,-47.932,179.296,6.235,149.335
C08004=1135.084,-29.617,-47.944,179.299,6.235,149.334
C08005=1135.079,-29.367,-47.955,179.301,6.236,149.334
C08006=1135.073,-29.119,-47.968,179.304,6.238,149.333
C08007=1135.068,-28.869,-47.979,179.306,6.238,149.333
C08008=1135.063,-28.619,-47.991,179.309,6.239,149.332
C08009=1135.057,-28.369,-48.003,179.311,6.240,149.332
C08010=1135.052,-28.119,-48.015,179.313,6.240,149.331
C08011=1135.048,-27.870,-48.027,179.316,6.241,149.331
C08012=1135.042,-27.620,-48.039,179.318,6.241,149.330
C08013=1135.037,-27.370,-48.050,179.320,6.242,149.329
C08014=1135.031,-27.120,-48.062,179.323,6.243,149.329
C08015=1135.027,-26.871,-48.074,179.325,6.243,149.328
C08016=1135.022,-26.621,-48.086,179.327,6.244,149.328
C08017=1135.016,-26.371,-48.098,179.330,6.245,149.327
C08018=1135.011,-26.122,-48.110,179.332,6.245,149.327
C08019=1135.006,-25.873,-48.122,179.334,6.246,149.326
C08020=1135.001,-25.623,-48.134,179.337,6.247,149.326
C08021=1134.995,-25.373,-48.146,179.339,6.247,149.325
C08022=1134.990,-25.103,-48.158,179.342,6.249,149.324
C08023=1134.984,-24.833,-48.171,179.344,6.249,149.324
C08024=1134.978,-24.563,-48.184,179.347,6.250,149.323
C08025=1134.973,-24.293,-48.198,179.349,6.251,149.323
C08026=1134.968,-24.043,-48.209,179.352,6.251,149.322
C08027=1134.962,-23.793,-48.221,179.354,6.252,149.322
C08028=1134.957,-23.544,-48.234,179.357,6.253,149.321
C08029=1134.952,-23.294,-48.246,179.359,6.254,149.320
C08030=1134.946,-23.044,-48.258,179.362,6.255,149.320
C08031=1134.941,-22.795,-48.270,179.364,6.255,149.320
C08032=1134.936,-22.545,-48.282,179.366,6.256,149.319
C08033=1134.932,-22.296,-48.294,179.369,6.256,149.318
C08034=1134.926,-22.046,-48.306,179.371,6.257,149.318
C08035=1134.921,-21.796,-48.318,179.373,6.258,149.317
C08036=1134.916,-21.547,-48.331,179.376,6.258,149.317
C08037=1134.910,-21.297,-48.342,179.378,6.259,149.316
C08038=1134.905,-21.047,-48.355,179.380,6.260,149.316
C08039=1134.900,-20.798,-48.367,179.383,6.260,149.315
C08040=1134.894,-20.548,-48.380,179.385,6.262,149.315
C08041=1134.889,-20.298,-48.391,179.388,6.263,149.314
C08042=1134.884,-20.049,-48.404,179.390,6.263,149.313
C08043=1134.878,-19.799,-48.416,179.393,6.264,149.313
C08044=1134.874,-19.549,-48.427,179.395,6.265,149.312
C08045=1134.869,-19.300,-48.440,179.397,6.265,149.312
C08046=1134.863,-19.051,-48.452,179.400,6.266,149.311
C08047=1134.858,-18.801,-48.464,179.402,6.267,149.311
C08048=1134.854,-18.551,-48.477,179.404,6.267,149.310
C08049=1134.848,-18.301,-48.489,179.407,6.269,149.310
C08050=1134.843,-18.052,-48.502,179.409,6.270,149.309
C08051=1134.838,-17.802,-48.514,179.412,6.270,149.309
C08052=1134.832,-17.552,-48.526,179.414,6.271,149.308
C08053=1134.827,-17.302,-48.538,179.416,6.272,149.308
C08054=1134.822,-17.053,-48.551,179.419,6.272,149.307
C08055=1134.816,-16.803,-48.563,179.421,6.273,149.306
C08056=1134.811,-16.554,-48.575,179.423,6.274,149.306
C08057=1134.806,-16.305,-48.588,179.426,6.274,149.305
C08058=1134.801,-16.055,-48.600,179.429,6.276,149.305
C08059=1134.796,-15.805,-48.613,179.431,6.276,149.304
C08060=1134.791,-15.555,-48.625,179.434,6.277,149.304
C08061=1134.786,-15.305,-48.637,179.436,6.278,149.303
C08062=1134.781,-15.056,-48.650,179.438,6.278,149.303
C08063=1134.775,-14.806,-48.662,179.441,6.279,149.302
C08064=1134.770,-14.557,-48.674,179.443,6.280,149.301
C08065=1134.765,-14.307,-48.687,179.446,6.281,149.301
C08066=1134.759,-14.057,-48.699,179.448,6.282,149.300
C08067=1134.754,-13.807,-48.712,179.451,6.282,149.300
C08068=1134.749,-13.558,-48.725,179.453,6.283,149.299
C08069=1134.744,-13.308,-48.737,179.455,6.284,149.299
C08070=1134.739,-13.059,-48.749,179.458,6.284,149.298
C08071=1134.733,-12.809,-48.762,179.460,6.285,149.298
C08072=1134.728,-12.560,-48.775,179.463,6.286,149.297
C08073=1134.723,-12.309,-48.787,179.465,6.287,149.297
C08074=1134.718,-12.060,-48.799,179.467,6.288,149.296
C08075=1134.713,-11.811,-48.812,179.470,6.288,149.295
C08076=1134.708,-11.561,-48.825,179.472,6.289,149.295
C08077=1134.702,-11.311,-48.837,179.474,6.290,149.294
C08078=1134.697,-11.062,-48.850,179.477,6.290,149.294
C08079=1134.692,-10.812,-48.863,179.480,6.292,149.293
C08080=1134.687,-10.562,-48.875,179.482,6.293,149.293
C08081=1134.682,-10.313,-48.888,179.485,6.293,149.292
C08082=1134.677,-10.063,-48.900,179.487,6.294,149.292
C08083=1134.671,-9.814,-48.912,179.489,6.295,149.291
C08084=1134.666,-9.564,-48.926,179.492,6.295,149.291
C08085=1134.661,-9.314,-48.939,179.494,6.297,149.290
C08086=1134.656,-9.065,-48.951,179.497,6.298,149.290
C08087=1134.651,-8.816,-48.964,179.499,6.298,149.289
C08088=1134.646,-8.566,-48.977,179.501,6.299,149.288
C08089=1134.640,-8.315,-48.989,179.504,6.300,149.288
C08090=1134.635,-8.066,-49.002,179.506,6.300,149.287
C08091=1134.630,-7.817,-49.014,179.509,6.302,149.287
C08092=1134.625,-7.567,-49.027,179.512,6.302,149.286
C08093=1134.620,-7.317,-49.040,179.514,6.303,149.286
C08094=1134.614,-7.068,-49.053,179.516,6.304,149.285
C08095=1134.609,-6.818,-49.066,179.519,6.304,149.284
C08096=1134.605,-6.568,-49.079,179.522,6.306,149.284
C08097=1134.600,-6.319,-49.091,179.524,6.306,149.284
C08098=1134.594,-6.069,-49.105,179.526,6.307,149.283
C08099=1134.589,-5.820,-49.117,179.529,6.308,149.282
C08100=1134.584,-5.570,-49.130,179.531,6.308,149.282
C08101=1134.579,-5.321,-49.143,179.534,6.310,149.281
C08102=1134.573,-5.071,-49.156,179.536,6.310,149.281
C08103=1134.569,-4.821,-49.169,179.538,6.311,149.280
C08104=1134.563,-4.571,-49.181,179.541,6.312,149.280
C08105=1134.558,-4.322,-49.195,179.543,6.312,149.279
C08106=1134.552,-4.073,-49.207,179.546,6.314,149.279
C08107=1134.548,-3.823,-49.220,179.549,6.314,149.278
C08108=1134.543,-3.574,-49.233,179.551,6.315,149.278
C08109=1134.537,-3.324,-49.246,179.553,6.316,149.277
C08110=1134.532,-3.074,-49.259,179.556,6.316,149.276
C08111=1134.527,-2.825,-49.272,179.558,6.318,149.276
C08112=1134.521,-2.575,-49.285,179.561,6.319,149.275
C08113=1134.517,-2.325,-49.298,179.563,6.319,149.275
C08114=1134.511,-2.075,-49.311,179.565,6.320,149.274
C08115=1134.506,-1.826,-49.324,179.568,6.321,149.274
C08116=1134.501,-1.576,-49.336,179.571,6.322,149.273
C08117=1134.496,-1.326,-49.350,179.573,6.323,149.273
C08118=1134.490,-1.077,-49.362,179.575,6.324,149.272
C08119=1134.486,-0.828,-49.376,179.578,6.324,149.272
C08120=1134.480,-0.578,-49.389,179.581,6.326,149.271
C08121=1134.475,-0.329,-49.402,179.583,6.326,149.271
C08122=1134.470,-0.078,-49.415,179.586,6.327,149.270
C08123=1134.465,0.171,-49.428,179.588,6.328,149.269
C08124=1134.460,0.421,-49.441,179.590,6.329,149.269
C08125=1134.454,0.671,-49.454,179.593,6.330,149.268
C08126=1134.450,0.940,-49.468,179.595,6.330,149.268
C08127=1134.443,1.209,-49.482,179.599,6.332,149.267
C08128=1134.438,1.479,-49.497,179.601,6.333,149.267
C08129=1134.433,1.748,-49.511,179.603,6.333,149.266
C08130=1134.427,1.998,-49.524,179.606,6.335,149.265
C08131=1134.422,2.247,-49.537,179.608,6.335,149.265
C08132=1134.417,2.497,-49.551,179.611,6.336,149.264
C08133=1134.412,2.746,-49.564,179.613,6.337,149.264
C08134=1134.407,2.997,-49.577,179.616,6.338,149.263
C08135=1134.402,3.246,-49.590,179.619,6.339,149.263
C08136=1134.397,3.496,-49.604,179.621,6.339,149.262
C08137=1134.391,3.745,-49.617,179.623,6.340,149.262
C08138=1134.386,3.994,-49.630,179.626,6.341,149.261
C08139=1134.381,4.245,-49.643,179.628,6.342,149.261
C08140=1134.376,4.494,-49.657,179.631,6.343,149.260
C08141=1134.371,4.744,-49.670,179.633,6.343,149.259
C08142=1134.365,4.993,-49.683,179.636,6.345,149.259
C08143=1134.361,5.243,-49.697,179.639,6.345,149.258
C08144=1134.355,5.492,-49.710,179.641,6.346,149.258
C08145=1134.351,5.742,-49.724,179.644,6.348,149.257
C08146=1134.345,5.991,-49.737,179.646,6.348,149.257
C08147=1134.340,6.241,-49.750,179.648,6.349,149.256
C08148=1134.335,6.490,-49.764,179.651,6.350,149.256
C08149=1134.330,6.741,-49.777,179.654,6.351,149.255
C08150=1134.325,6.990,-49.790,179.656,6.352,149.255
C08151=1134.320,7.240,-49.804,179.658,6.353,149.254
C08152=1134.314,7.489,-49.817,179.661,6.354,149.253
C08153=1134.310,7.739,-49.831,179.664,6.355,149.253
C08154=1134.304,7.988,-49.844,179.666,6.356,149.253
C08155=1134.299,8.238,-49.858,179.668,6.356,149.252
C08156=1134.294,8.487,-49.871,179.671,6.358,149.251
C08157=1134.289,8.737,-49.885,179.673,6.358,149.251
C08158=1134.283,8.986,-49.898,179.676,6.359,149.250
C08159=1134.278,9.237,-49.911,179.679,6.360,149.250
C08160=1134.273,9.485,-49.925,179.681,6.361,149.249
C08161=1134.268,9.736,-49.938,179.684,6.362,149.249
C08162=1134.263,9.985,-49.952,179.686,6.362,149.248
C08163=1134.258,10.235,-49.965,179.689,6.364,149.248
C08164=1134.253,10.484,-49.979,179.691,6.364,149.247
C08165=1134.248,10.733,-49.993,179.693,6.365,149.247
C08166=1134.242,10.983,-50.006,179.696,6.367,149.246
C08167=1134.237,11.232,-50.020,179.699,6.367,149.245
C08168=1134.232,11.482,-50.034,179.701,6.368,149.245
C08169=1134.227,11.731,-50.047,179.704,6.370,149.245
C08170=1134.222,11.982,-50.061,179.707,6.370,149.244
C08171=1134.217,12.231,-50.075,179.709,6.371,149.243
C08172=1134.212,12.480,-50.088,179.711,6.373,149.243
C08173=1134.207,12.730,-50.102,179.714,6.373,149.242
C08174=1134.202,12.980,-50.116,179.716,6.374,149.242
C08175=1134.196,13.229,-50.129,179.718,6.375,149.241
C08176=1134.191,13.479,-50.143,179.722,6.376,149.241
C08177=1134.187,13.728,-50.157,179.724,6.377,149.240
C08178=1134.181,13.978,-50.170,179.726,6.377,149.240
C08179=1134.176,14.228,-50.184,179.729,6.379,149.239
C08180=1134.171,14.476,-50.198,179.731,6.380,149.239
C08181=1134.166,14.727,-50.211,179.734,6.380,149.238
C08182=1134.161,14.976,-50.226,179.737,6.382,149.237
C08183=1134.155,15.225,-50.240,179.739,6.382,149.237
C08184=1134.151,15.475,-50.252,179.741,6.383,149.236
C08185=1134.146,15.725,-50.267,179.745,6.384,149.236
C08186=1134.140,15.974,-50.281,179.747,6.385,149.235
C08187=1134.135,16.224,-50.295,179.749,6.386,149.235
C08188=1134.130,16.474,-50.309,179.752,6.387,149.234
C08189=1134.125,16.723,-50.322,179.754,6.388,149.234
C08190=1134.120,16.973,-50.336,179.757,6.390,149.233
C08191=1134.115,17.222,-50.350,179.760,6.390,149.233
C08192=1134.109,17.472,-50.364,179.762,6.391,149.232
C08193=1134.104,17.722,-50.378,179.765,6.393,149.232
C08194=1134.099,17.971,-50.392,179.767,6.393,149.231
C08195=1134.094,18.220,-50.406,179.769,6.394,149.231
C08196=1134.090,18.470,-50.420,179.772,6.395,149.230
C08197=1134.084,18.720,-50.433,179.775,6.396,149.229
C08198=1134.079,18.969,-50.447,179.777,6.397,149.229
C08199=1134.074,19.219,-50.461,179.780,6.398,149.228
C08200=1134.069,19.469,-50.476,179.782,6.399,149.228
C08201=1134.063,19.718,-50.490,179.785,6.399,149.227
C08202=1134.058,19.967,-50.504,179.787,6.401,149.227
C08203=1134.053,20.217,-50.518,179.790,6.402,149.226
C08204=1134.048,20.467,-50.531,179.793,6.403,149.226
C08205=1134.043,20.716,-50.546,179.795,6.404,149.225
C08206=1134.038,20.966,-50.559,179.798,6.404,149.225
C08207=1134.033,21.215,-50.574,179.800,6.406,149.224
C08208=1134.028,21.464,-50.588,179.803,6.407,149.224
C08209=1134.023,21.714,-50.602,179.805,6.407,149.223
C08210=1134.018,21.964,-50.616,179.808,6.409,149.223
C08211=1134.013,22.214,-50.630,179.810,6.410,149.222
C08212=1134.007,22.463,-50.644,179.813,6.411,149.221
C08213=1134.002,22.712,-50.659,179.816,6.412,149.221
C08214=1133.998,22.962,-50.673,179.818,6.413,149.220
C08215=1133.993,23.212,-50.687,179.821,6.414,149.220
C08216=1133.987,23.461,-50.701,179.823,6.415,149.219
C08217=1133.982,23.710,-50.715,179.826,6.416,149.219
C08218=1133.977,23.960,-50.730,179.829,6.417,149.218
C08219=1133.972,24.210,-50.744,179.831,6.417,149.218
C08220=1133.967,24.459,-50.758,179.834,6.419,149.217
C08221=1133.962,24.709,-50.772,179.836,6.419,149.217
C08222=1133.957,24.958,-50.786,179.839,6.421,149.216
C08223=1133.952,25.208,-50.801,179.841,6.422,149.216
C08224=1133.947,25.458,-50.815,179.844,6.422,149.215
C08225=1133.941,25.707,-50.829,179.847,6.424,149.215
C08226=1133.936,25.956,-50.843,179.849,6.425,149.214
C08227=1133.931,26.206,-50.857,179.852,6.426,149.213
C08228=1133.926,26.455,-50.873,179.854,6.427,149.213
C08229=1133.921,26.705,-50.887,179.856,6.428,149.213
C08230=1133.916,26.975,-50.902,179.860,6.429,149.212
C08231=1133.910,27.243,-50.918,179.862,6.431,149.211
C08232=1133.904,27.512,-50.933,179.865,6.431,149.211
C08233=1133.899,27.781,-50.948,179.868,6.433,149.210
C08234=1133.894,28.031,-50.963,179.870,6.433,149.210
C08235=1133.889,28.281,-50.977,179.873,6.435,149.209
C08236=1133.884,28.530,-50.992,179.875,6.435,149.209
C08237=1133.879,28.779,-51.007,179.879,6.437,149.208
C08238=1133.873,29.028,-51.021,179.881,6.437,149.208
C08239=1133.868,29.278,-51.035,179.883,6.438,149.207
C08240=1133.864,29.528,-51.049,179.886,6.440,149.206
C08241=1133.858,29.777,-51.065,179.888,6.440,149.206
C08242=1133.853,30.027,-51.079,179.891,6.442,149.206
C08243=1133.848,30.277,-51.093,179.894,6.442,149.205
C08244=1133.843,30.526,-51.108,179.897,6.444,149.204
C08245=1133.839,30.776,-51.123,179.899,6.445,149.204
C08246=1133.833,31.025,-51.136,179.902,6.446,149.203
C08247=1133.827,31.275,-51.151,179.904,6.447,149.203
C08248=1133.823,31.524,-51.166,179.906,6.448,149.202
C08249=1133.818,31.773,-51.181,179.909,6.449,149.202
C08250=1133.813,32.023,-51.195,179.912,6.450,149.201
C08251=1133.808,32.272,-51.210,179.914,6.451,149.201
C08252=1133.802,32.522,-51.225,179.917,6.452,149.200
C08253=1133.798,32.772,-51.239,179.920,6.453,149.200
C08254=1133.793,33.021,-51.254,179.922,6.454,149.199
C08255=1133.788,33.271,-51.268,179.925,6.456,149.199
C08256=1133.782,33.521,-51.283,179.927,6.456,149.198
C08257=1133.778,33.770,-51.298,179.930,6.458,149.198
C08258=1133.773,34.020,-51.312,179.932,6.459,149.197
C08259=1133.768,34.269,-51.327,179.936,6.460,149.196
C08260=1133.762,34.518,-51.342,179.938,6.461,149.196
C08261=1133.757,34.768,-51.356,179.940,6.462,149.196
C08262=1133.752,35.017,-51.371,179.943,6.463,149.195
C08263=1133.746,35.267,-51.386,179.945,6.464,149.194
C08264=1133.742,35.516,-51.401,179.948,6.465,149.194
C08265=1133.737,35.766,-51.415,179.950,6.466,149.194
C08266=1133.731,36.015,-51.431,179.954,6.467,149.193
C08267=1133.726,36.265,-51.445,179.956,6.468,149.192
C08268=1133.722,36.514,-51.460,179.959,6.470,149.192
C08269=1133.716,36.764,-51.475,179.961,6.470,149.191
C08270=1133.711,37.013,-51.490,179.964,6.472,149.191
C08271=1133.707,37.263,-51.504,179.966,6.473,149.190
C08272=1133.701,37.512,-51.520,179.969,6.474,149.190
C08273=1133.696,37.762,-51.534,179.971,6.475,149.189
C08274=1133.691,38.011,-51.550,179.974,6.476,149.189
C08275=1133.686,38.261,-51.564,179.977,6.477,149.188
C08276=1133.681,38.510,-51.579,179.980,6.479,149.188
C08277=1133.675,38.760,-51.594,179.982,6.479,149.187
C08278=1133.671,39.009,-51.609,179.985,6.481,149.187
C08279=1133.665,39.259,-51.624,179.987,6.481,149.186
C08280=1133.660,39.508,-51.639,179.990,6.483,149.186
C08281=1133.656,39.758,-51.654,179.992,6.484,149.185
C08282=1133.651,40.008,-51.669,179.995,6.485,149.185
C08283=1133.646,40.257,-51.684,179.998,6.486,149.184
C08284=1133.641,40.506,-51.700,-180.000,6.488,149.184
C08285=1133.636,40.756,-51.714,-179.997,6.488,149.183
C08286=1133.630,41.006,-51.729,-179.994,6.490,149.183
C08287=1133.626,41.255,-51.744,-179.992,6.491,149.182
C08288=1133.620,41.505,-51.759,-179.989,6.492,149.181
C08289=1133.615,41.754,-51.774,-179.987,6.493,149.181
C08290=1133.611,42.003,-51.789,-179.984,6.494,149.180
C08291=1133.605,42.253,-51.804,-179.981,6.496,149.180
C08292=1133.600,42.502,-51.819,-179.979,6.496,149.179
C08293=1133.595,42.751,-51.835,-179.976,6.498,149.179
C08294=1133.591,43.001,-51.850,-179.974,6.499,149.178
C08295=1133.585,43.251,-51.865,-179.970,6.500,149.178
C08296=1133.580,43.501,-51.881,-179.968,6.501,149.177
C08297=1133.575,43.750,-51.896,-179.965,6.502,149.177
C08298=1133.570,43.999,-51.911,-179.963,6.503,149.176
C08299=1133.565,44.249,-51.925,-179.960,6.505,149.176
C08300=1133.559,44.498,-51.941,-179.958,6.505,149.175
C08301=1133.555,44.747,-51.956,-179.955,6.507,149.175
C08302=1133.550,44.997,-51.972,-179.952,6.507,149.174
C08303=1133.545,45.246,-51.987,-179.950,6.509,149.174
C08304=1133.540,45.496,-52.002,-179.947,6.511,149.173
C08305=1133.534,45.746,-52.017,-179.944,6.511,149.173
C08306=1133.530,45.995,-52.032,-179.942,6.513,149.172
C08307=1133.524,46.244,-52.048,-179.939,6.514,149.172
C08308=1133.520,46.494,-52.063,-179.937,6.515,149.171
C08309=1133.515,46.744,-52.079,-179.934,6.516,149.171
C08310=1133.509,46.993,-52.095,-179.931,6.517,149.170
C08311=1133.505,47.242,-52.110,-179.929,6.518,149.170
C08312=1133.499,47.492,-52.124,-179.926,6.519,149.169
C08313=1133.495,47.742,-52.140,-179.923,6.521,149.169
C08314=1133.490,47.991,-52.155,-179.921,6.522,149.168
C08315=1133.484,48.241,-52.171,-179.918,6.524,149.168
C08316=1133.480,48.490,-52.186,-179.915,6.524,149.167
C08317=1133.474,48.739,-52.202,-179.913,6.526,149.167
C08318=1133.469,48.989,-52.217,-179.911,6.526,149.166
C08319=1133.465,49.238,-52.232,-179.907,6.528,149.166
C08320=1133.459,49.488,-52.248,-179.905,6.529,149.165
C08321=1133.454,49.737,-52.264,-179.902,6.530,149.165
C08322=1133.450,49.987,-52.279,-179.900,6.532,149.164
C08323=1133.445,50.236,-52.295,-179.897,6.532,149.164
C08324=1133.439,50.486,-52.310,-179.894,6.534,149.163
C08325=1133.434,50.735,-52.326,-179.891,6.535,149.163
C08326=1133.430,50.985,-52.341,-179.889,6.536,149.162
C08327=1133.424,51.234,-52.357,-179.886,6.538,149.162
C08328=1133.419,51.484,-52.372,-179.884,6.538,149.161
C08329=1133.414,51.733,-52.387,-179.881,6.540,149.161
C08330=1133.410,51.982,-52.404,-179.878,6.541,149.160
C08331=1133.405,52.232,-52.420,-179.876,6.542,149.160
C08332=1133.399,52.481,-52.435,-179.873,6.544,149.159
C08333=1133.394,52.731,-52.451,-179.870,6.544,149.158
C08334=1133.390,52.999,-52.468,-179.868,6.546,149.158
C08335=1133.384,53.268,-52.485,-179.865,6.547,149.158
C08336=1133.378,53.537,-52.501,-179.862,6.549,149.157
C08337=1133.373,53.805,-52.518,-179.859,6.550,149.156
C08338=1133.367,54.055,-52.533,-179.856,6.551,149.156
C08339=1133.363,54.304,-52.550,-179.853,6.552,149.155
C08340=1133.358,54.553,-52.565,-179.851,6.553,149.155
C08341=1133.353,54.803,-52.581,-179.848,6.555,149.154
C08342=1133.348,55.053,-52.597,-179.845,6.556,149.154
C08343=1133.342,55.302,-52.612,-179.843,6.557,149.153
C08344=1133.337,55.551,-52.629,-179.840,6.559,149.153
C08345=1133.333,55.801,-52.645,-179.838,6.560,149.152
C08346=1133.327,56.051,-52.660,-179.835,6.561,149.152
C08347=1133.323,56.300,-52.675,-179.832,6.562,149.151
C08348=1133.318,56.549,-52.692,-179.830,6.563,149.151
C08349=1133.313,56.799,-52.707,-179.827,6.565,149.150
C08350=1133.307,57.048,-52.723,-179.824,6.566,149.150
C08351=1133.303,57.298,-52.739,-179.822,6.567,149.149
C08352=1133.297,57.547,-52.755,-179.819,6.569,149.149
C08353=1133.292,57.796,-52.771,-179.816,6.570,149.148
C08354=1133.287,58.046,-52.787,-179.814,6.571,149.148
C08355=1133.282,58.295,-52.803,-179.811,6.572,149.147
C08356=1133.277,58.545,-52.819,-179.808,6.574,149.147
C08357=1133.272,58.795,-52.835,-179.806,6.574,149.146
C08358=1133.267,59.043,-52.851,-179.803,6.576,149.146
C08359=1133.263,59.293,-52.866,-179.800,6.578,149.145
C08360=1133.258,59.542,-52.883,-179.798,6.579,149.145
C08361=1133.253,59.792,-52.898,-179.795,6.580,149.144
C08362=1133.248,60.042,-52.914,-179.792,6.581,149.144
C08363=1133.243,60.291,-52.931,-179.790,6.582,149.143
C08364=1133.238,60.540,-52.946,-179.787,6.584,149.143
C08365=1133.233,60.789,-52.963,-179.784,6.585,149.142
C08366=1133.228,61.039,-52.979,-179.782,6.586,149.142
C08367=1133.223,61.288,-52.995,-179.779,6.588,149.141
C08368=1133.218,61.538,-53.011,-179.776,6.589,149.141
C08369=1133.213,61.787,-53.027,-179.773,6.590,149.140
C08370=1133.208,62.037,-53.043,-179.771,6.591,149.140
C08371=1133.203,62.286,-53.059,-179.768,6.593,149.139
C08372=1133.198,62.536,-53.076,-179.766,6.594,149.139
C08373=1133.192,62.785,-53.092,-179.763,6.595,149.138
C08374=1133.188,63.035,-53.108,-179.760,6.597,149.138
C08375=1133.183,63.284,-53.125,-179.758,6.598,149.137
C08376=1133.177,63.533,-53.140,-179.755,6.599,149.137
C08377=1133.173,63.783,-53.157,-179.752,6.601,149.136
C08378=1133.167,64.032,-53.172,-179.750,6.601,149.136
C08379=1133.163,64.282,-53.189,-179.747,6.603,149.135
C08380=1133.158,64.531,-53.205,-179.744,6.605,149.135
C08381=1133.153,64.781,-53.221,-179.741,6.605,149.134
C08382=1133.148,65.029,-53.238,-179.739,6.607,149.134
C08383=1133.143,65.280,-53.254,-179.736,6.608,149.133
C08384=1133.138,65.529,-53.271,-179.733,6.610,149.133
C08385=1133.133,65.778,-53.287,-179.730,6.611,149.132
C08386=1133.128,66.028,-53.303,-179.728,6.612,149.132
C08387=1133.123,66.277,-53.319,-179.725,6.614,149.132
C08388=1133.119,66.526,-53.336,-179.723,6.615,149.131
C08389=1133.113,66.776,-53.352,-179.720,6.616,149.130
C08390=1133.109,67.025,-53.368,-179.717,6.618,149.130
C08391=1133.103,67.274,-53.385,-179.715,6.618,149.130
C08392=1133.098,67.525,-53.401,-179.712,6.620,149.129
C08393=1133.094,67.774,-53.418,-179.709,6.621,149.128
C08394=1133.088,68.023,-53.434,-179.706,6.623,149.128
C08395=1133.084,68.272,-53.451,-179.704,6.624,149.128
C08396=1133.078,68.522,-53.467,-179.701,6.625,149.127
C08397=1133.073,68.772,-53.484,-179.698,6.627,149.127
C08398=1133.068,69.020,-53.500,-179.695,6.628,149.126
C08399=1133.064,69.270,-53.517,-179.693,6.629,149.126
C08400=1133.058,69.520,-53.533,-179.690,6.631,149.125
C08401=1133.053,69.769,-53.549,-179.687,6.633,149.125
C08402=1133.049,70.018,-53.566,-179.685,6.633,149.124
C08403=1133.044,70.267,-53.582,-179.682,6.635,149.124
C08404=1133.038,70.517,-53.600,-179.679,6.636,149.123
C08405=1133.034,70.767,-53.616,-179.676,6.638,149.123
C08406=1133.029,71.016,-53.632,-179.674,6.639,149.122
C08407=1133.024,71.265,-53.649,-179.671,6.640,149.122
C08408=1133.019,71.515,-53.666,-179.668,6.642,149.121
C08409=1133.014,71.764,-53.682,-179.666,6.643,149.121
C08410=1133.009,72.013,-53.699,-179.663,6.644,149.120
C08411=1133.003,72.263,-53.716,-179.660,6.645,149.120
C08412=1132.999,72.512,-53.732,-179.657,6.647,149.119
C08413=1132.995,72.762,-53.749,-179.655,6.649,149.119
C08414=1132.989,73.011,-53.766,-179.653,6.650,149.118
C08415=1132.984,73.260,-53.783,-179.650,6.651,149.118
C08416=1132.980,73.510,-53.799,-179.647,6.653,149.117
C08417=1132.974,73.759,-53.816,-179.644,6.654,149.117
C08418=1132.969,74.008,-53.833,-179.642,6.655,149.116
C08419=1132.964,74.258,-53.850,-179.639,6.657,149.116
C08420=1132.959,74.507,-53.866,-179.636,6.658,149.116
C08421=1132.955,74.756,-53.883,-179.633,6.660,149.115
C08422=1132.949,75.006,-53.900,-179.630,6.661,149.115
C08423=1132.945,75.256,-53.917,-179.628,6.662,149.114
C08424=1132.939,75.505,-53.934,-179.625,6.664,149.114
C08425=1132.935,75.754,-53.951,-179.623,6.665,149.113
C08426=1132.930,76.004,-53.967,-179.619,6.667,149.113
C08427=1132.924,76.253,-53.984,-179.617,6.668,149.112
C08428=1132.920,76.502,-54.001,-179.614,6.669,149.112
C08429=1132.915,76.752,-54.018,-179.612,6.671,149.111
C08430=1132.910,77.001,-54.035,-179.609,6.672,149.111
C08431=1132.904,77.251,-54.052,-179.606,6.674,149.110
C08432=1132.900,77.500,-54.068,-179.604,6.675,149.110
C08433=1132.895,77.750,-54.086,-179.601,6.676,149.109
C08434=1132.891,77.999,-54.103,-179.598,6.678,149.109
C08435=1132.885,78.248,-54.120,-179.595,6.680,149.108
C08436=1132.880,78.497,-54.137,-179.592,6.681,149.108
C08437=1132.875,78.747,-54.154,-179.590,6.682,149.107
C08438=1132.870,79.016,-54.172,-179.587,6.683,149.107
C08439=1132.864,79.284,-54.190,-179.584,6.685,149.106
C08440=1132.860,79.552,-54.208,-179.581,6.686,149.106
C08441=1132.854,79.821,-54.227,-179.578,6.688,149.105
C08442=1132.849,80.070,-54.245,-179.576,6.690,149.105
C08443=1132.844,80.319,-54.261,-179.572,6.691,149.104
C08444=1132.839,80.569,-54.279,-179.570,6.693,149.104
C08445=1132.834,80.818,-54.295,-179.567,6.694,149.104
C08446=1132.829,81.067,-54.313,-179.564,6.696,149.103
C08447=1132.825,81.316,-54.330,-179.562,6.697,149.103
C08448=1132.819,81.566,-54.347,-179.559,6.698,149.102
C08449=1132.815,81.815,-54.365,-179.556,6.700,149.102
C08450=1132.810,82.065,-54.382,-179.553,6.701,149.101
C08451=1132.804,82.314,-54.398,-179.551,6.703,149.101
C08452=1132.800,82.563,-54.416,-179.548,6.704,149.100
C08453=1132.795,82.813,-54.433,-179.546,6.705,149.100
C08454=1132.790,83.062,-54.450,-179.542,6.707,149.099
C08455=1132.785,83.311,-54.468,-179.540,6.708,149.099
C08456=1132.780,83.561,-54.485,-179.537,6.710,149.098
C08457=1132.775,83.811,-54.502,-179.534,6.712,149.098
C08458=1132.770,84.059,-54.519,-179.532,6.713,149.098
C08459=1132.765,84.309,-54.537,-179.529,6.714,149.097
C08460=1132.760,84.558,-54.554,-179.526,6.715,149.096
C08461=1132.756,84.807,-54.571,-179.523,6.717,149.096
C08462=1132.750,85.057,-54.588,-179.521,6.719,149.096
C08463=1132.745,85.306,-54.606,-179.518,6.720,149.095
C08464=1132.741,85.556,-54.623,-179.515,6.722,149.095
C08465=1132.736,85.805,-54.641,-179.513,6.723,149.094
C08466=1132.731,86.055,-54.658,-179.510,6.724,149.094
C08467=1132.726,86.304,-54.676,-179.507,6.726,149.093
C08468=1132.721,86.553,-54.693,-179.504,6.728,149.093
C08469=1132.716,86.802,-54.711,-179.502,6.729,149.092
C08470=1132.711,87.052,-54.728,-179.499,6.731,149.092
C08471=1132.706,87.301,-54.746,-179.496,6.733,149.092
C08472=1132.701,87.550,-54.762,-179.493,6.733,149.091
C08473=1132.696,87.800,-54.780,-179.491,6.735,149.090
C08474=1132.692,88.049,-54.798,-179.488,6.736,149.090
C08475=1132.686,88.299,-54.816,-179.485,6.738,149.090
C08476=1132.682,88.548,-54.833,-179.482,6.740,149.089
C08477=1132.677,88.797,-54.850,-179.480,6.741,149.089
C08478=1132.672,89.046,-54.868,-179.476,6.743,149.088
C08479=1132.667,89.296,-54.886,-179.474,6.744,149.088
C08480=1132.662,89.545,-54.904,-179.471,6.746,149.087
C08481=1132.658,89.794,-54.921,-179.469,6.747,149.087
C08482=1132.653,90.043,-54.939,-179.466,6.748,149.086
C08483=1132.648,90.293,-54.956,-179.463,6.750,149.086
C08484=1132.643,90.542,-54.974,-179.461,6.752,149.086
C08485=1132.638,90.792,-54.992,-179.457,6.753,149.085
C08486=1132.633,91.041,-55.009,-179.455,6.755,149.085
C08487=1132.628,91.291,-55.027,-179.452,6.756,149.084
C08488=1132.623,91.539,-55.045,-179.449,6.758,149.084
C08489=1132.618,91.789,-55.062,-179.446,6.760,149.083
C08490=1132.613,92.038,-55.080,-179.444,6.761,149.083
C08491=1132.608,92.288,-55.098,-179.442,6.762,149.082
C08492=1132.603,92.537,-55.116,-179.438,6.763,149.082
C08493=1132.599,92.786,-55.134,-179.436,6.765,149.081
C08494=1132.593,93.036,-55.151,-179.433,6.767,149.081
C08495=1132.588,93.285,-55.169,-179.430,6.768,149.081
C08496=1132.584,93.534,-55.187,-179.427,6.770,149.080
C08497=1132.579,93.783,-55.205,-179.425,6.772,149.080
C08498=1132.574,94.032,-55.223,-179.422,6.773,149.079
C08499=1132.568,94.282,-55.240,-179.419,6.775,149.079
C08500=1132.564,94.531,-55.258,-179.416,6.776,149.078
C08501=1132.559,94.781,-55.277,-179.413,6.778,149.078
C08502=1132.554,95.030,-55.295,-179.411,6.779,149.077
C08503=1132.549,95.280,-55.313,-179.408,6.781,149.077
C08504=1132.545,95.529,-55.331,-179.406,6.782,149.077
C08505=1132.540,95.778,-55.349,-179.403,6.784,149.076
C08506=1132.535,96.027,-55.367,-179.400,6.786,149.076
C08507=1132.529,96.277,-55.384,-179.397,6.787,149.075
C08508=1132.525,96.526,-55.402,-179.394,6.789,149.075
C08509=1132.520,96.775,-55.420,-179.391,6.790,149.074
C08510=1132.515,97.025,-55.438,-179.389,6.792,149.074
C08511=1132.510,97.274,-55.456,-179.386,6.794,149.073
C08512=1132.506,97.524,-55.474,-179.383,6.795,149.073
C08513=1132.501,97.773,-55.492,-179.380,6.797,149.073
C08514=1132.496,98.022,-55.510,-179.378,6.799,149.072
C08515=1132.491,98.271,-55.528,-179.375,6.800,149.072
C08516=1132.486,98.520,-55.546,-179.372,6.802,149.071
C08517=1132.481,98.769,-55.564,-179.369,6.803,149.071
C08518=1132.477,99.019,-55.582,-179.366,6.805,149.070
C08519=1132.471,99.269,-55.601,-179.363,6.806,149.070
C08520=1132.466,99.517,-55.620,-179.361,6.808,149.069
C08521=1132.461,99.767,-55.638,-179.359,6.809,149.069
C08522=1132.457,100.016,-55.656,-179.356,6.811,149.069
C08523=1132.452,100.266,-55.674,-179.353,6.812,149.068
C08524=1132.447,100.515,-55.692,-179.350,6.814,149.068
C08525=1132.442,100.764,-55.710,-179.348,6.816,149.067
C08526=1132.437,101.013,-55.729,-179.345,6.817,149.067
C08527=1132.432,101.263,-55.747,-179.342,6.819,149.066
C08528=1132.428,101.512,-55.765,-179.339,6.820,149.066
C08529=1132.423,101.761,-55.784,-179.336,6.822,149.065
C08530=1132.418,102.010,-55.802,-179.333,6.824,149.065
C08531=1132.413,102.259,-55.820,-179.331,6.825,149.065
C08532=1132.407,102.509,-55.838,-179.328,6.827,149.064
C08533=1132.403,102.759,-55.856,-179.325,6.829,149.064
C08534=1132.399,103.007,-55.875,-179.322,6.830,149.063
C08535=1132.394,103.256,-55.893,-179.320,6.832,149.063
C08536=1132.388,103.506,-55.912,-179.317,6.834,149.063
C08537=1132.384,103.756,-55.930,-179.314,6.835,149.062
C08538=1132.379,104.004,-55.949,-179.312,6.837,149.062
C08539=1132.374,104.254,-55.967,-179.308,6.838,149.061
C08540=1132.369,104.503,-55.985,-179.306,6.840,149.061
C08541=1132.364,104.753,-56.004,-179.303,6.842,149.060
C08542=1132.359,105.021,-56.024,-179.300,6.843,149.060
C08543=1132.354,105.289,-56.044,-179.297,6.846,149.059
C08544=1132.349,105.557,-56.063,-179.294,6.847,149.059
C08545=1132.343,105.826,-56.083,-179.291,6.849,149.058
C08546=1132.339,106.075,-56.102,-179.288,6.850,149.058
C08547=1132.334,106.324,-56.120,-179.285,6.852,149.058
C08548=1132.328,106.573,-56.140,-179.283,6.854,149.057
C08549=1132.324,106.823,-56.158,-179.280,6.855,149.057
C08550=1132.319,107.072,-56.176,-179.277,6.857,149.056
C08551=1132.314,107.321,-56.195,-179.274,6.859,149.056
C08552=1132.310,107.571,-56.213,-179.272,6.860,149.055
C08553=1132.305,107.820,-56.232,-179.269,6.862,149.055
C08554=1132.299,108.069,-56.251,-179.266,6.864,149.055
C08555=1132.295,108.319,-56.269,-179.263,6.865,149.054
C08556=1132.290,108.568,-56.288,-179.261,6.867,149.054
C08557=1132.285,108.817,-56.306,-179.258,6.869,149.053
C08558=1132.281,109.066,-56.325,-179.255,6.870,149.053
C08559=1132.275,109.316,-56.344,-179.252,6.873,149.053
C08560=1132.271,109.565,-56.363,-179.249,6.874,149.052
C08561=1132.265,109.815,-56.382,-179.246,6.876,149.052
C08562=1132.261,110.063,-56.400,-179.243,6.878,149.051
C08563=1132.256,110.313,-56.420,-179.241,6.879,149.051
C08564=1132.251,110.562,-56.438,-179.238,6.881,149.050
C08565=1132.246,110.811,-56.457,-179.235,6.883,149.050
C08566=1132.242,111.061,-56.476,-179.232,6.884,149.050
C08567=1132.237,111.309,-56.494,-179.230,6.886,149.049
C08568=1132.232,111.559,-56.513,-179.227,6.888,149.049
C08569=1132.227,111.808,-56.532,-179.224,6.889,149.048
C08570=1132.222,112.057,-56.551,-179.221,6.891,149.048
C08571=1132.217,112.307,-56.570,-179.219,6.893,149.047
C08572=1132.212,112.555,-56.589,-179.216,6.894,149.047
C08573=1132.208,112.805,-56.609,-179.213,6.896,149.047
C08574=1132.203,113.054,-56.626,-179.210,6.898,149.046
C08575=1132.198,113.304,-56.646,-179.208,6.899,149.046
C08576=1132.193,113.552,-56.665,-179.204,6.902,149.045
C08577=1132.188,113.803,-56.684,-179.202,6.904,149.045
C08578=1132.184,114.051,-56.702,-179.199,6.905,149.045
C08579=1132.178,114.300,-56.722,-179.196,6.907,149.044
C08580=1132.174,114.550,-56.740,-179.193,6.909,149.044
C08581=1132.169,114.799,-56.759,-179.191,6.910,149.043
C08582=1132.164,115.048,-56.779,-179.188,6.912,149.043
C08583=1132.159,115.297,-56.798,-179.185,6.914,149.043
C08584=1132.155,115.546,-56.817,-179.183,6.915,149.042
C08585=1132.149,115.796,-56.836,-179.180,6.917,149.042
C08586=1132.145,116.045,-56.855,-179.177,6.919,149.041
C08587=1132.140,116.294,-56.874,-179.174,6.920,149.041
C08588=1132.136,116.543,-56.893,-179.171,6.923,149.041
C08589=1132.130,116.792,-56.913,-179.168,6.924,149.040
C08590=1132.125,117.042,-56.932,-179.166,6.926,149.040
C08591=1132.121,117.291,-56.950,-179.163,6.928,149.039
C08592=1132.116,117.540,-56.970,-179.160,6.929,149.039
C08593=1132.110,117.789,-56.989,-179.157,6.931,149.039
C08594=1132.107,118.030,-57.008,-179.155,6.933,149.038
C08595=1132.102,118.272,-57.026,-179.152,6.935,149.038
C08596=1132.097,118.513,-57.046,-179.149,6.936,149.037
C08597=1132.073,119.724,-57.140,-179.807,8.266,149.529
C08598=1132.069,119.973,-57.161,-179.805,8.269,149.530
C08599=1132.064,120.222,-57.180,-179.803,8.273,149.530
C08600=1132.059,120.471,-57.200,-179.801,8.277,149.530
C08601=1132.054,120.720,-57.220,-179.800,8.279,149.531
C08602=1132.050,120.970,-57.240,-179.798,8.283,149.531
C08603=1132.044,121.218,-57.259,-179.796,8.286,149.531
C08604=1132.040,121.467,-57.279,-179.794,8.290,149.531
C08605=1132.035,121.717,-57.299,-179.792,8.294,149.532
C08606=1132.030,121.966,-57.319,-179.791,8.297,149.532
C08607=1132.025,122.215,-57.339,-179.789,8.300,149.532
C08608=1132.021,122.464,-57.358,-179.787,8.304,149.532
C08609=1132.016,122.714,-57.378,-179.785,8.307,149.532
C08610=1132.011,122.963,-57.398,-179.784,8.310,149.533
C08611=1132.007,123.212,-57.418,-179.781,8.314,149.533
C08612=1132.002,123.461,-57.438,-179.779,8.317,149.533
C08613=1131.997,123.710,-57.458,-179.777,8.321,149.534
C08614=1131.992,123.960,-57.477,-179.776,8.324,149.534
C08615=1131.988,124.209,-57.498,-179.774,8.327,149.534
C08616=1131.982,124.458,-57.517,-179.772,8.331,149.534
C08617=1131.978,124.707,-57.537,-179.770,8.334,149.535
C08618=1131.973,124.956,-57.557,-179.769,8.337,149.535
C08619=1131.969,125.205,-57.577,-179.767,8.341,149.535
C08620=1131.964,125.455,-57.597,-179.765,8.344,149.536
C08621=1131.960,125.704,-57.617,-179.764,8.347,149.536
C08622=1131.954,125.952,-57.637,-179.761,8.350,149.536
C08623=1131.950,126.201,-57.657,-179.760,8.354,149.536
C08624=1131.945,126.451,-57.677,-179.758,8.357,149.537
C08625=1131.940,126.700,-57.698,-179.756,8.361,149.537
C08626=1131.936,126.949,-57.718,-179.754,8.364,149.537
C08627=1131.931,127.199,-57.738,-179.753,8.367,149.537
C08628=1131.926,127.447,-57.758,-179.751,8.371,149.538
C08629=1131.921,127.697,-57.777,-179.749,8.374,149.538
C08630=1131.917,127.945,-57.798,-179.748,8.377,149.538
C08631=1131.911,128.195,-57.819,-179.746,8.381,149.539
C08632=1131.907,128.444,-57.838,-179.744,8.384,149.539
C08633=1131.902,128.693,-57.859,-179.743,8.387,149.539
C08634=1131.898,128.942,-57.879,-179.740,8.390,149.539
C08635=1131.892,129.191,-57.899,-179.739,8.394,149.540
C08636=1131.887,129.440,-57.919,-179.737,8.397,149.540
C08637=1131.883,129.689,-57.940,-179.735,8.401,149.540
C08638=1131.875,130.101,-57.973,-179.732,8.406,149.541
C08639=1131.868,130.513,-58.007,-179.730,8.411,149.541
C08640=1131.860,130.926,-58.040,-179.727,8.417,149.542
C08641=1131.851,131.337,-58.073,-179.724,8.423,149.542
C08642=1131.847,131.586,-58.094,-179.723,8.425,149.542
C08643=1131.841,131.836,-58.114,-179.721,8.429,149.543
C08644=1131.837,132.085,-58.134,-179.720,8.432,149.543
C08645=1131.833,132.334,-58.155,-179.718,8.435,149.543
C08646=1131.827,132.583,-58.176,-179.716,8.439,149.543
C08647=1131.823,132.832,-58.196,-179.715,8.442,149.544
C08648=1131.819,133.081,-58.217,-179.712,8.446,149.544
C08649=1131.813,133.331,-58.237,-179.711,8.449,149.545
C08650=1131.809,133.580,-58.257,-179.709,8.452,149.545
C08651=1131.804,133.829,-58.278,-179.708,8.455,149.545
C08652=1131.799,134.078,-58.299,-179.706,8.459,149.545
C08653=1131.795,134.327,-58.319,-179.705,8.461,149.546
C08654=1131.790,134.576,-58.339,-179.703,8.465,149.546
C08655=1131.785,134.825,-58.360,-179.702,8.468,149.546
C08656=1131.781,135.074,-58.381,-179.700,8.471,149.547
C08657=1131.776,135.323,-58.401,-179.698,8.475,149.547
C08658=1131.771,135.573,-58.421,-179.697,8.478,149.547
C08659=1131.766,135.822,-58.442,-179.695,8.482,149.548
C08660=1131.761,136.071,-58.463,-179.694,8.485,149.548
C08661=1131.757,136.320,-58.483,-179.691,8.488,149.548
C08662=1131.752,136.569,-58.503,-179.690,8.491,149.548
C08663=1131.747,136.818,-58.524,-179.688,8.495,149.549
C08664=1131.743,137.067,-58.545,-179.687,8.498,149.549
C08665=1131.737,137.316,-58.566,-179.685,8.501,149.549
C08666=1131.733,137.565,-58.586,-179.684,8.504,149.550
C08667=1131.728,137.815,-58.607,-179.682,8.508,149.550
C08668=1131.723,138.064,-58.627,-179.681,8.511,149.550
C08669=1131.719,138.313,-58.648,-179.680,8.514,149.551
C08670=1131.714,138.561,-58.669,-179.678,8.518,149.551
C08671=1131.710,138.810,-58.690,-179.677,8.520,149.551
C08672=1131.704,139.059,-58.711,-179.675,8.524,149.552
C08673=1131.700,139.308,-58.731,-179.674,8.527,149.552
C08674=1131.695,139.558,-58.752,-179.672,8.531,149.552
C08675=1131.691,139.807,-58.773,-179.670,8.533,149.553
C08676=1131.686,140.057,-58.794,-179.669,8.537,149.553
C08677=1131.681,140.306,-58.814,-179.667,8.540,149.553
C08678=1131.676,140.555,-58.835,-179.666,8.544,149.554
C08679=1131.672,140.803,-58.856,-179.664,8.547,149.554
C08680=1131.667,141.052,-58.877,-179.663,8.550,149.554
C08681=1131.662,141.302,-58.898,-179.662,8.554,149.555
C08682=1131.657,141.551,-58.919,-179.660,8.556,149.555
C08683=1131.652,141.800,-58.939,-179.659,8.560,149.555
C08684=1131.648,142.049,-58.960,-179.657,8.563,149.556
C08685=1131.643,142.298,-58.982,-179.655,8.567,149.556
C08686=1131.639,142.547,-59.002,-179.654,8.570,149.557
C08687=1131.634,142.796,-59.023,-179.653,8.573,149.557
C08688=1131.629,143.045,-59.044,-179.651,8.576,149.557
C08689=1131.624,143.294,-59.065,-179.650,8.579,149.558
C08690=1131.620,143.509,-59.084,-179.649,8.582,149.558
C08691=1131.616,143.723,-59.101,-179.648,8.585,149.558
C08692=1131.612,143.939,-59.119,-179.646,8.588,149.559
C08693=1131.608,144.153,-59.137,-179.645,8.591,149.559
C08694=1131.604,144.368,-59.155,-179.644,8.594,149.559
C08695=1131.600,144.583,-59.174,-179.643,8.596,149.559
C08696=1131.596,144.798,-59.192,-179.642,8.600,149.560
C08697=1131.592,145.013,-59.210,-179.640,8.602,149.560
C08698=1131.588,145.261,-59.231,-179.637,8.607,149.560
C08699=1131.583,145.510,-59.252,-179.635,8.610,149.561
C08700=1131.577,145.760,-59.273,-179.632,8.614,149.561
C08701=1131.573,146.008,-59.294,-179.629,8.618,149.561
C08702=1131.569,146.258,-59.316,-179.627,8.622,149.561
C08703=1131.563,146.507,-59.337,-179.624,8.626,149.561
C08704=1131.559,146.756,-59.358,-179.621,8.631,149.561
C08705=1131.554,147.005,-59.379,-179.618,8.635,149.562
C08706=1131.549,147.253,-59.400,-179.615,8.639,149.562
C08707=1131.545,147.503,-59.422,-179.613,8.642,149.562
C08708=1131.540,147.752,-59.443,-179.610,8.646,149.562
C08709=1131.535,148.001,-59.464,-179.607,8.650,149.562
C08710=1131.531,148.250,-59.485,-179.604,8.655,149.562
C08711=1131.526,148.500,-59.507,-179.601,8.659,149.562
C08712=1131.521,148.748,-59.528,-179.599,8.662,149.563
C08713=1131.517,148.997,-59.549,-179.596,8.666,149.563
C08714=1131.512,149.247,-59.571,-179.593,8.670,149.563
C08715=1131.508,149.495,-59.592,-179.591,8.673,149.563
C08716=1131.502,149.744,-59.613,-179.588,8.678,149.563
C08717=1131.497,149.993,-59.635,-179.585,8.681,149.563
C08718=1131.493,150.243,-59.656,-179.582,8.686,149.563
C08719=1131.488,150.492,-59.678,-179.580,8.689,149.563
C08720=1131.484,150.740,-59.699,-179.577,8.693,149.564
C08721=1131.479,150.990,-59.721,-179.574,8.697,149.564
C08722=1131.474,151.239,-59.742,-179.572,8.700,149.564
C08723=1131.470,151.487,-59.764,-179.569,8.704,149.564
C08724=1131.465,151.737,-59.786,-179.566,8.708,149.564
C08725=1131.460,151.986,-59.807,-179.563,8.712,149.564
C08726=1131.455,152.234,-59.829,-179.561,8.716,149.564
C08727=1131.451,152.484,-59.851,-179.558,8.719,149.564
C08728=1131.446,152.732,-59.872,-179.555,8.723,149.565
C08729=1131.441,152.982,-59.893,-179.553,8.726,149.565
C08730=1131.437,153.231,-59.915,-179.550,8.730,149.565
C08731=1131.432,153.480,-59.937,-179.548,8.734,149.565
C08732=1131.428,153.729,-59.959,-179.544,8.738,149.565
C08733=1131.423,153.978,-59.981,-179.542,8.741,149.565
C08734=1131.418,154.226,-60.002,-179.539,8.745,149.565
C08735=1131.413,154.476,-60.024,-179.537,8.748,149.565
C08736=1131.408,154.725,-60.045,-179.534,8.752,149.565
C08737=1131.404,154.974,-60.068,-179.531,8.756,149.565
C08738=1131.399,155.223,-60.089,-179.529,8.760,149.566
C08739=1131.394,155.472,-60.111,-179.526,8.763,149.566
C08740=1131.390,155.721,-60.133,-179.523,8.767,149.566
C08741=1131.385,155.970,-60.155,-179.521,8.770,149.566
C08742=1131.381,156.219,-60.177,-179.518,8.774,149.566
C08743=1131.376,156.467,-60.198,-179.515,8.777,149.566
C08744=1131.372,156.717,-60.220,-179.513,8.781,149.566
C08745=1131.366,156.966,-60.243,-179.510,8.785,149.566
C08746=1131.362,157.180,-60.262,-179.508,8.787,149.566
C08747=1131.358,157.395,-60.280,-179.506,8.790,149.567
C08748=1131.354,157.610,-60.300,-179.504,8.794,149.567
C08749=1131.350,157.824,-60.319,-179.501,8.797,149.567
C08750=1131.346,158.039,-60.337,-179.499,8.799,149.567
C08751=1131.342,158.254,-60.356,-179.497,8.802,149.567
C08752=1131.338,158.468,-60.376,-179.495,8.806,149.567
C08753=1131.334,158.683,-60.394,-179.492,8.809,149.567
C08754=1131.330,158.932,-60.416,-179.489,8.812,149.567
C08755=1131.325,159.181,-60.438,-179.487,8.815,149.567
C08756=1131.321,159.429,-60.460,-179.485,8.818,149.567
C08757=1131.316,159.679,-60.483,-179.482,8.822,149.567
C08758=1131.311,159.928,-60.505,-179.479,8.825,149.567
C08759=1131.307,160.177,-60.527,-179.477,8.829,149.568
C08760=1131.302,160.426,-60.549,-179.475,8.832,149.568
C08761=1131.298,160.674,-60.571,-179.471,8.836,149.568
C08762=1131.293,160.924,-60.594,-179.469,8.839,149.568
C08763=1131.288,161.173,-60.616,-179.467,8.842,149.568
C08764=1131.284,161.422,-60.638,-179.464,8.846,149.568
C08765=1131.278,161.670,-60.661,-179.462,8.849,149.568
C08766=1131.274,161.920,-60.683,-179.459,8.853,149.568
C08767=1131.270,162.169,-60.705,-179.457,8.856,149.568
C08768=1131.265,162.417,-60.727,-179.454,8.859,149.568
C08769=1131.260,162.667,-60.750,-179.451,8.862,149.568
C08770=1131.255,162.915,-60.771,-179.449,8.866,149.569
C08771=1131.251,163.164,-60.794,-179.447,8.869,149.569
C08772=1131.246,163.414,-60.817,-179.444,8.872,149.569
C08773=1131.241,163.662,-60.839,-179.442,8.875,149.569
C08774=1131.238,163.911,-60.861,-179.439,8.879,149.569
C08775=1131.233,164.161,-60.884,-179.437,8.882,149.569
C08776=1131.228,164.409,-60.906,-179.434,8.886,149.569
C08777=1131.223,164.658,-60.929,-179.432,8.889,149.569
C08778=1131.219,164.907,-60.952,-179.429,8.892,149.569
C08779=1131.214,165.156,-60.973,-179.427,8.895,149.569
C08780=1131.209,165.405,-60.997,-179.424,8.898,149.569
C08781=1131.205,165.654,-61.019,-179.422,8.901,149.569
C08782=1131.200,165.902,-61.042,-179.419,8.905,149.569
C08783=1131.196,166.152,-61.064,-179.417,8.908,149.570
C08784=1131.191,166.401,-61.087,-179.415,8.911,149.570
C08785=1131.186,166.649,-61.109,-179.412,8.914,149.570
C08786=1131.182,166.898,-61.132,-179.410,8.917,149.570
C08787=1131.177,167.148,-61.154,-179.407,8.920,149.570
C08788=1131.172,167.396,-61.177,-179.405,8.924,149.570
C08789=1131.167,167.645,-61.199,-179.403,8.927,149.570
C08790=1131.164,167.894,-61.222,-179.400,8.930,149.570
C08791=1131.159,168.143,-61.245,-179.397,8.933,149.570
C08792=1131.154,168.392,-61.267,-179.395,8.937,149.570
C08793=1131.149,168.641,-61.291,-179.394,8.939,149.570
C08794=1131.145,168.890,-61.314,-179.391,8.942,149.570
C08795=1131.140,169.139,-61.336,-179.388,8.945,149.570
C08796=1131.135,169.388,-61.359,-179.386,8.949,149.571
C08797=1131.131,169.636,-61.382,-179.384,8.952,149.571
C08798=1131.126,169.886,-61.404,-179.381,8.955,149.571
C08799=1131.122,170.135,-61.427,-179.379,8.958,149.571
C08800=1131.117,170.383,-61.450,-179.376,8.961,149.571
C08801=1131.112,170.633,-61.473,-179.375,8.964,149.571
C08802=1131.109,170.847,-61.493,-179.372,8.967,149.571
C08803=1131.104,171.061,-61.512,-179.370,8.969,149.571
C08804=1131.100,171.276,-61.532,-179.369,8.972,149.571
C08805=1131.096,171.490,-61.552,-179.366,8.975,149.571
C08806=1131.092,171.705,-61.572,-179.365,8.978,149.571
C08807=1131.088,171.919,-61.591,-179.363,8.980,149.571
C08808=1131.084,172.134,-61.611,-179.361,8.982,149.571
C08809=1131.081,172.349,-61.631,-179.358,8.985,149.571
C08810=1131.075,172.597,-61.654,-179.357,8.988,149.572
C08811=1131.071,172.846,-61.676,-179.354,8.991,149.572
C08812=1131.067,173.095,-61.700,-179.352,8.994,149.572
C08813=1131.062,173.345,-61.723,-179.349,8.997,149.572
C08814=1131.058,173.593,-61.746,-179.348,9.000,149.572
C08815=1131.053,173.842,-61.769,-179.345,9.003,149.572
C08816=1131.048,174.091,-61.792,-179.343,9.006,149.572
C08817=1131.044,174.339,-61.815,-179.341,9.010,149.572
C08818=1131.039,174.588,-61.838,-179.339,9.012,149.572
C08819=1131.034,174.837,-61.862,-179.336,9.015,149.572
C08820=1131.030,175.086,-61.885,-179.334,9.018,149.572
C08821=1131.026,175.335,-61.908,-179.332,9.021,149.573
C08822=1131.021,175.584,-61.931,-179.330,9.024,149.573
C08823=1131.016,175.832,-61.954,-179.327,9.027,149.573
C08824=1131.011,176.082,-61.977,-179.326,9.030,149.573
C08825=1131.007,176.330,-62.000,-179.323,9.033,149.573
C08826=1131.002,176.579,-62.024,-179.321,9.036,149.573
C08827=1130.998,176.828,-62.047,-179.319,9.039,149.573
C08828=1130.993,177.077,-62.070,-179.317,9.042,149.573
C08829=1130.988,177.326,-62.094,-179.314,9.045,149.573
C08830=1130.984,177.575,-62.116,-179.313,9.048,149.574
C08831=1130.980,177.824,-62.140,-179.310,9.051,149.574
C08832=1130.975,178.073,-62.163,-179.308,9.053,149.574
C08833=1130.970,178.322,-62.186,-179.306,9.057,149.574
C08834=1130.966,178.571,-62.210,-179.304,9.060,149.574
C08835=1130.961,178.820,-62.233,-179.302,9.062,149.574
C08836=1130.957,179.068,-62.256,-179.300,9.066,149.574
C08837=1130.952,179.317,-62.280,-179.297,9.069,149.574
C08838=1130.947,179.566,-62.303,-179.293,9.072,149.574
C08839=1130.943,179.815,-62.326,-179.291,9.075,149.574
C08840=1130.938,180.064,-62.350,-179.288,9.079,149.574
C08841=1130.933,180.312,-62.374,-179.284,9.083,149.574
C08842=1130.929,180.561,-62.397,-179.282,9.086,149.574
C08843=1130.924,180.810,-62.420,-179.279,9.090,149.574
C08844=1130.919,181.059,-62.444,-179.276,9.092,149.574
C08845=1130.915,181.308,-62.468,-179.272,9.096,149.574
C08846=1130.911,181.556,-62.491,-179.269,9.099,149.574
C08847=1130.906,181.805,-62.514,-179.266,9.103,149.574
C08848=1130.902,182.054,-62.537,-179.264,9.106,149.574
C08849=1130.897,182.303,-62.561,-179.260,9.109,149.574
C08850=1130.893,182.553,-62.585,-179.258,9.113,149.574
C08851=1130.889,182.801,-62.609,-179.255,9.116,149.574
C08852=1130.884,183.050,-62.633,-179.252,9.119,149.574
C08853=1130.879,183.299,-62.656,-179.249,9.122,149.574
C08854=1130.875,183.548,-62.680,-179.247,9.125,149.574
C08855=1130.870,183.797,-62.703,-179.244,9.129,149.574
C08856=1130.865,184.045,-62.728,-179.241,9.131,149.574
C08857=1130.860,184.294,-62.751,-179.239,9.134,149.574
C08858=1130.857,184.509,-62.772,-179.236,9.137,149.574
C08859=1130.853,184.722,-62.792,-179.234,9.140,149.574
C08860=1130.849,184.937,-62.813,-179.231,9.143,149.574
C08861=1130.845,185.152,-62.834,-179.229,9.145,149.574
C08862=1130.841,185.366,-62.854,-179.227,9.148,149.574
C08863=1130.837,185.581,-62.874,-179.225,9.150,149.574
C08864=1130.833,185.795,-62.894,-179.222,9.153,149.574
C08865=1130.829,186.010,-62.915,-179.220,9.156,149.574
C08866=1130.825,186.258,-62.939,-179.217,9.158,149.574
C08867=1130.821,186.508,-62.963,-179.215,9.162,149.574
C08868=1130.815,186.756,-62.987,-179.213,9.164,149.574
C08869=1130.811,187.005,-63.011,-179.210,9.167,149.574
C08870=1130.806,187.254,-63.035,-179.208,9.170,149.574
C08871=1130.802,187.502,-63.059,-179.205,9.173,149.574
C08872=1130.797,187.751,-63.082,-179.204,9.176,149.574
C08873=1130.793,188.000,-63.106,-179.201,9.179,149.574
C08874=1130.788,188.249,-63.131,-179.198,9.182,149.574
C08875=1130.784,188.498,-63.155,-179.197,9.184,149.574
C08876=1130.779,188.747,-63.179,-179.194,9.187,149.574
C08877=1130.775,188.995,-63.203,-179.192,9.190,149.574
C08878=1130.770,189.244,-63.226,-179.190,9.193,149.574
C08879=1130.765,189.493,-63.251,-179.188,9.195,149.574
C08880=1130.761,189.742,-63.275,-179.185,9.198,149.574
C08881=1130.757,189.990,-63.299,-179.183,9.200,149.574
C08882=1130.752,190.239,-63.323,-179.181,9.204,149.574
C08883=1130.747,190.488,-63.347,-179.179,9.206,149.574
C08884=1130.743,190.736,-63.372,-179.177,9.209,149.574
C08885=1130.739,190.986,-63.396,-179.175,9.212,149.575
C08886=1130.733,191.235,-63.420,-179.173,9.214,149.575
C08887=1130.729,191.483,-63.444,-179.171,9.216,149.575
C08888=1130.725,191.732,-63.468,-179.170,9.219,149.575
C08889=1130.719,191.980,-63.493,-179.167,9.222,149.575
C08890=1130.716,192.230,-63.517,-179.165,9.224,149.575
C08891=1130.711,192.478,-63.541,-179.164,9.227,149.575
C08892=1130.707,192.727,-63.565,-179.162,9.230,149.575
C08893=1130.701,192.976,-63.589,-179.160,9.232,149.575
C08894=1130.698,193.225,-63.614,-179.159,9.235,149.575
C08895=1130.692,193.474,-63.638,-179.157,9.237,149.575
C08896=1130.688,193.722,-63.662,-179.155,9.240,149.576
C08897=1130.684,193.970,-63.687,-179.153,9.242,149.576
C08898=1130.679,194.220,-63.712,-179.152,9.245,149.576
C08899=1130.675,194.468,-63.736,-179.150,9.247,149.576
C08900=1130.670,194.717,-63.759,-179.148,9.250,149.576
C08901=1130.665,194.966,-63.784,-179.147,9.252,149.577
C08902=1130.661,195.215,-63.808,-179.145,9.255,149.577
C08903=1130.656,195.464,-63.833,-179.144,9.257,149.577
C08904=1130.652,195.712,-63.857,-179.142,9.260,149.577
C08905=1130.648,195.961,-63.881,-179.141,9.262,149.577
C08906=1130.643,196.210,-63.906,-179.140,9.265,149.577
C08907=1130.638,196.459,-63.930,-179.136,9.268,149.577
C08908=1130.634,196.708,-63.955,-179.132,9.272,149.577
C08909=1130.629,196.956,-63.979,-179.128,9.277,149.577
C08910=1130.625,197.205,-64.003,-179.124,9.280,149.577
C08911=1130.620,197.454,-64.028,-179.120,9.284,149.577
C08912=1130.616,197.703,-64.052,-179.116,9.288,149.576
C08913=1130.611,197.951,-64.077,-179.112,9.292,149.576
C08914=1130.607,198.165,-64.098,-179.109,9.295,149.576
C08915=1130.603,198.380,-64.119,-179.105,9.298,149.576
C08916=1130.600,198.594,-64.141,-179.102,9.301,149.576
C08917=1130.595,198.809,-64.162,-179.099,9.305,149.576
C08918=1130.591,199.023,-64.184,-179.096,9.307,149.576
C08919=1130.588,199.237,-64.205,-179.092,9.311,149.575
C08920=1130.584,199.451,-64.226,-179.089,9.314,149.575
C08921=1130.580,199.665,-64.247,-179.086,9.316,149.575
C08922=1130.576,199.915,-64.272,-179.083,9.320,149.575
C08923=1130.571,200.163,-64.296,-179.079,9.323,149.575
C08924=1130.566,200.412,-64.321,-179.076,9.327,149.575
C08925=1130.562,200.661,-64.347,-179.072,9.330,149.575
C08926=1130.558,200.909,-64.371,-179.068,9.334,149.574
C08927=1130.553,201.158,-64.396,-179.065,9.337,149.574
C08928=1130.548,201.407,-64.421,-179.061,9.341,149.574
C08929=1130.545,201.656,-64.446,-179.058,9.344,149.574
C08930=1130.539,201.904,-64.470,-179.055,9.347,149.574
C08931=1130.535,202.153,-64.496,-179.052,9.350,149.574
C08932=1130.531,202.402,-64.520,-179.048,9.353,149.574
C08933=1130.527,202.650,-64.546,-179.045,9.356,149.573
C08934=1130.521,202.899,-64.571,-179.042,9.360,149.573
C08935=1130.518,203.148,-64.596,-179.039,9.362,149.573
C08936=1130.513,203.396,-64.621,-179.035,9.366,149.573
C08937=1130.509,203.645,-64.646,-179.032,9.369,149.573
C08938=1130.503,203.894,-64.671,-179.029,9.371,149.573
C08939=1130.500,204.142,-64.696,-179.026,9.374,149.573
C08940=1130.495,204.391,-64.721,-179.023,9.378,149.573
C08941=1130.491,204.640,-64.746,-179.020,9.381,149.572
C08942=1130.485,204.889,-64.771,-179.017,9.383,149.572
C08943=1130.482,205.137,-64.796,-179.014,9.386,149.572
C08944=1130.477,205.386,-64.821,-179.012,9.389,149.572
C08945=1130.473,205.635,-64.847,-179.009,9.392,149.572
C08946=1130.468,205.883,-64.871,-179.006,9.395,149.572
C08947=1130.463,206.132,-64.897,-179.003,9.398,149.572
C08948=1130.459,206.381,-64.923,-179.000,9.401,149.572
C08949=1130.455,206.629,-64.947,-178.998,9.403,149.572
C08950=1130.450,206.878,-64.973,-178.995,9.406,149.572
C08951=1130.446,207.126,-64.998,-178.992,9.408,149.572
C08952=1130.441,207.376,-65.023,-178.990,9.412,149.572
C08953=1130.436,207.624,-65.049,-178.988,9.414,149.572
C08954=1130.432,207.873,-65.074,-178.985,9.417,149.572
C08955=1130.427,208.122,-65.099,-178.983,9.419,149.572
C08956=1130.423,208.370,-65.125,-178.981,9.422,149.572
C08957=1130.418,208.619,-65.150,-178.978,9.424,149.572
C08958=1130.414,208.868,-65.176,-178.976,9.427,149.572
C08959=1130.410,209.116,-65.200,-178.974,9.429,149.572
C08960=1130.406,209.365,-65.226,-178.971,9.433,149.572
C08961=1130.401,209.613,-65.251,-178.969,9.435,149.572
C08962=1130.397,209.862,-65.277,-178.968,9.437,149.572
C08963=1130.392,210.111,-65.303,-178.965,9.440,149.572
C08964=1130.387,210.359,-65.328,-178.963,9.443,149.572
C08965=1130.383,210.608,-65.353,-178.961,9.445,149.572
C08966=1130.379,210.857,-65.379,-178.959,9.447,149.572
C08967=1130.374,211.105,-65.404,-178.957,9.450,149.572
C08968=1130.370,211.354,-65.430,-178.956,9.452,149.572
C08969=1130.365,211.603,-65.456,-178.953,9.455,149.572
C08970=1130.361,211.817,-65.478,-178.952,9.457,149.572
C08971=1130.358,212.031,-65.500,-178.950,9.459,149.572
C08972=1130.353,212.245,-65.522,-178.949,9.461,149.573
C08973=1130.350,212.460,-65.543,-178.948,9.464,149.573
C08974=1130.346,212.674,-65.566,-178.947,9.466,149.573
C08975=1130.342,212.888,-65.588,-178.945,9.468,149.573
C08976=1130.338,213.102,-65.610,-178.944,9.470,149.573
C08977=1130.334,213.316,-65.632,-178.942,9.472,149.573
C08978=1130.330,213.565,-65.658,-178.941,9.475,149.573
C08979=1130.325,213.814,-65.683,-178.939,9.478,149.574
C08980=1130.321,214.062,-65.709,-178.937,9.480,149.574
C08981=1130.316,214.311,-65.735,-178.936,9.483,149.574
C08982=1130.312,214.559,-65.760,-178.933,9.486,149.574
C08983=1130.308,214.808,-65.786,-178.932,9.488,149.574
C08984=1130.303,215.056,-65.811,-178.930,9.491,149.574
C08985=1130.299,215.305,-65.837,-178.928,9.494,149.575
C08986=1130.295,215.554,-65.863,-178.926,9.496,149.575
C08987=1130.290,215.803,-65.889,-178.924,9.499,149.575
C08988=1130.285,216.051,-65.915,-178.922,9.502,149.575
C08989=1130.281,216.300,-65.940,-178.920,9.505,149.575
C08990=1130.276,216.549,-65.966,-178.918,9.508,149.575
C08991=1130.272,216.798,-65.992,-178.916,9.510,149.575
C08992=1130.267,217.046,-66.017,-178.914,9.514,149.575
C08993=1130.263,217.294,-66.043,-178.911,9.517,149.576
C08994=1130.259,217.543,-66.069,-178.910,9.519,149.576
C08995=1130.254,217.792,-66.096,-178.907,9.522,149.576
C08996=1130.250,218.041,-66.122,-178.905,9.526,149.576
C08997=1130.245,218.289,-66.147,-178.902,9.529,149.576
C08998=1130.241,218.537,-66.173,-178.900,9.531,149.576
C08999=1130.237,218.786,-66.198,-178.898,9.534,149.576
C09000=1130.232,219.035,-66.226,-178.895,9.538,149.576
C09001=1130.228,219.284,-66.251,-178.893,9.541,149.576
C09002=1130.223,219.532,-66.277,-178.891,9.544,149.576
C09003=1130.219,219.780,-66.302,-178.888,9.547,149.577
C09004=1130.215,220.029,-66.328,-178.886,9.550,149.577
C09005=1130.210,220.278,-66.355,-178.883,9.553,149.577
C09006=1130.206,220.527,-66.381,-178.881,9.557,149.577
C09007=1130.201,220.775,-66.406,-178.878,9.560,149.577
C09008=1130.197,221.023,-66.432,-178.876,9.563,149.577
C09009=1130.192,221.272,-66.459,-178.873,9.566,149.577
C09010=1130.188,221.521,-66.485,-178.871,9.569,149.577
C09011=1130.183,221.770,-66.511,-178.867,9.573,149.577
C09012=1130.179,222.018,-66.538,-178.865,9.576,149.577
C09013=1130.175,222.267,-66.563,-178.862,9.579,149.577
C09014=1130.170,222.514,-66.590,-178.859,9.582,149.577
C09015=1130.165,222.763,-66.616,-178.856,9.586,149.577
C09016=1130.161,223.012,-66.642,-178.854,9.589,149.577
C09017=1130.157,223.260,-66.668,-178.851,9.592,149.577
C09018=1130.152,223.510,-66.695,-178.848,9.595,149.577
C09019=1130.148,223.758,-66.721,-178.845,9.599,149.577
C09020=1130.144,224.007,-66.747,-178.842,9.602,149.577
C09021=1130.139,224.255,-66.774,-178.839,9.605,149.577
C09022=1130.135,224.504,-66.800,-178.836,9.609,149.577
C09023=1130.130,224.752,-66.827,-178.833,9.612,149.577
C09024=1130.126,225.001,-66.852,-178.830,9.616,149.577
C09025=1130.121,225.249,-66.879,-178.826,9.619,149.577
C09026=1130.117,225.464,-66.901,-178.824,9.622,149.577
C09027=1130.114,225.677,-66.924,-178.821,9.625,149.577
C09028=1130.110,225.892,-66.947,-178.818,9.628,149.577
C09029=1130.106,226.105,-66.970,-178.815,9.631,149.577
C09030=1130.103,226.320,-66.993,-178.813,9.634,149.577
C09031=1130.099,226.534,-67.015,-178.810,9.637,149.577
C09032=1130.095,226.748,-67.038,-178.807,9.640,149.577
C09033=1130.091,226.962,-67.061,-178.804,9.643,149.577
C09034=1130.086,227.210,-67.088,-178.801,9.646,149.577
C09035=1130.082,227.459,-67.114,-178.797,9.650,149.577
C09036=1130.078,227.708,-67.141,-178.793,9.653,149.576
C09037=1130.074,227.956,-67.167,-178.790,9.657,149.576
C09038=1130.069,228.204,-67.194,-178.786,9.660,149.576
C09039=1130.065,228.453,-67.220,-178.783,9.664,149.576
C09040=1130.060,228.702,-67.247,-178.779,9.667,149.576
C09041=1130.055,228.950,-67.274,-178.776,9.671,149.576
C09042=1130.051,229.198,-67.301,-178.772,9.674,149.576
C09043=1130.047,229.448,-67.327,-178.768,9.677,149.575
C09044=1130.043,229.696,-67.353,-178.764,9.681,149.575
C09045=1130.038,229.944,-67.380,-178.761,9.685,149.575
C09046=1130.033,230.193,-67.407,-178.757,9.688,149.575
C09047=1130.030,230.442,-67.434,-178.753,9.691,149.575
C09048=1130.025,230.690,-67.461,-178.750,9.695,149.575
C09049=1130.021,230.939,-67.488,-178.746,9.698,149.575
C09050=1130.016,231.187,-67.515,-178.742,9.701,149.574
C09051=1130.012,231.435,-67.542,-178.738,9.705,149.574
C09052=1130.007,231.684,-67.569,-178.735,9.708,149.574
C09053=1130.003,231.932,-67.596,-178.732,9.711,149.574
C09054=1129.999,232.180,-67.623,-178.728,9.715,149.574
C09055=1129.994,232.429,-67.650,-178.725,9.717,149.573
C09056=1129.990,232.678,-67.677,-178.721,9.721,149.573
C09057=1129.985,232.927,-67.704,-178.718,9.723,149.573
C09058=1129.982,233.175,-67.731,-178.715,9.727,149.573
C09059=1129.977,233.423,-67.758,-178.712,9.730,149.573
C09060=1129.972,233.672,-67.785,-178.708,9.733,149.573
C09061=1129.968,233.920,-67.812,-178.705,9.736,149.573
C09062=1129.964,234.169,-67.839,-178.702,9.739,149.573
C09063=1129.960,234.418,-67.866,-178.699,9.741,149.572
C09064=1129.955,234.666,-67.893,-178.695,9.745,149.572
C09065=1129.951,234.914,-67.920,-178.693,9.747,149.572
C09066=1129.946,235.163,-67.948,-178.690,9.750,149.572
C09067=1129.942,235.412,-67.975,-178.687,9.753,149.572
C09068=1129.937,235.660,-68.002,-178.684,9.756,149.572
C09069=1129.933,235.908,-68.030,-178.681,9.758,149.572
C09070=1129.929,236.156,-68.056,-178.678,9.761,149.571
C09071=1129.925,236.405,-68.084,-178.675,9.764,149.571
C09072=1129.920,236.654,-68.111,-178.672,9.767,149.571
C09073=1129.916,236.902,-68.139,-178.669,9.770,149.571
C09074=1129.911,237.150,-68.166,-178.667,9.772,149.571
C09075=1129.907,237.399,-68.193,-178.664,9.774,149.571
C09076=1129.903,237.648,-68.220,-178.661,9.777,149.571
C09077=1129.898,237.896,-68.248,-178.659,9.779,149.571
C09078=1129.894,238.144,-68.275,-178.656,9.782,149.571
C09079=1129.890,238.393,-68.303,-178.653,9.785,149.571
C09080=1129.885,238.641,-68.330,-178.651,9.787,149.570
C09081=1129.880,238.890,-68.357,-178.649,9.790,149.571
C09082=1129.877,239.104,-68.381,-178.646,9.792,149.570
C09083=1129.873,239.318,-68.405,-178.644,9.794,149.570
C09084=1129.869,239.531,-68.428,-178.642,9.796,149.570
C09085=1129.866,239.746,-68.451,-178.641,9.798,149.570
C09086=1129.862,239.960,-68.476,-178.638,9.800,149.570
C09087=1129.858,240.173,-68.499,-178.637,9.802,149.570
C09088=1129.854,240.388,-68.523,-178.635,9.804,149.570
C09089=1129.851,240.601,-68.547,-178.632,9.806,149.570
C09090=1129.846,240.850,-68.574,-178.630,9.809,149.570
C09091=1129.842,241.098,-68.601,-178.628,9.811,149.570
C09092=1129.838,241.347,-68.629,-178.626,9.813,149.570
C09093=1129.833,241.595,-68.656,-178.624,9.815,149.570
C09094=1129.829,241.843,-68.684,-178.622,9.818,149.570
C09095=1129.825,242.092,-68.712,-178.620,9.820,149.570
C09096=1129.820,242.341,-68.740,-178.618,9.822,149.570
C09097=1129.816,242.588,-68.768,-178.616,9.824,149.570
C09098=1129.811,242.838,-68.795,-178.614,9.827,149.570
C09099=1129.807,243.086,-68.823,-178.613,9.829,149.570
C09100=1129.803,243.335,-68.850,-178.611,9.831,149.570
C09101=1129.799,243.583,-68.878,-178.609,9.834,149.570
C09102=1129.794,243.831,-68.905,-178.607,9.836,149.571
C09103=1129.790,244.080,-68.933,-178.606,9.838,149.571
C09104=1129.786,244.328,-68.961,-178.604,9.840,149.571
C09105=1129.781,244.576,-68.988,-178.602,9.843,149.571
C09106=1129.777,244.825,-69.017,-178.601,9.844,149.571
C09107=1129.772,245.073,-69.045,-178.599,9.847,149.571
